// DE-BOUNCE TIMER FOR GL8 CASE STOP2 IS RAISED SWITCH OFF
GVL_CONVEYORS.GL8.CaseStop2IsRaisedTimerOff (IN := GVL_CONVEYORS.GL8.Case_Stop_Load_2_Extended_Right AND GVL_CONVEYORS.GL8.Case_Stop_Load_2_Extended_Left , PT := T#500MS);
GVL_CONVEYORS.GL8.CaseStop2IsRaisedTimerOffDoneBit := GVL_CONVEYORS.GL8.CaseStop2IsRaisedTimerOff.Q;
GVL_CONVEYORS.GL8.CaseStop2IsRaisedTimerOffElapsedTime := GVL_CONVEYORS.GL8.CaseStop2IsRaisedTimerOff.ET;
GVL_CONVEYORS.GL8.CaseStop2RaisedSwitchIsOff := GVL_CONVEYORS.GL8.CaseStop2IsRaisedTimerOffDoneBit;

END_PROGRAM

// ---- Machine System/PRGs/Conveyors/MOTOR_FAULTS.TcPOU
PROGRAM MOTOR_FAULTS
VAR
	TON_GL1_MTR: TON; // MOTOR FAULT DELAY TIMER
	TON_GL2_MTR: TON; // MOTOR FAULT DELAY TIMER
	TON_GL3_MTR: TON; // MOTOR FAULT DELAY TIMER
	TON_GL4_MTR: TON; // MOTOR FAULT DELAY TIMER
	TON_GL5A_MTR: TON; // MOTOR FAULT DELAY TIMER
	TON_GL5B_MTR: TON; // MOTOR FAULT DELAY TIMER
	TON_GL6_MTR: TON; // MOTOR FAULT DELAY TIMER
	TON_GL7_MTR: TON; // MOTOR FAULT DELAY TIMER
	TON_GL8_MTR: TON; // MOTOR FAULT DELAY TIMER
	TON_GL9_MTR: TON; // MOTOR FAULT DELAY TIMER
	TON_GL10_MTR: TON; // MOTOR FAULT DELAY TIMER
	TON_GL11_MTR: TON; // MOTOR FAULT DELAY TIMER
	
	GL1_MTR: sClearPath;
	GL2_MTR: sClearPath;
	GL3_MTR: sClearPath;
	GL4_MTR: sClearPath;
	GL5_MTR: sClearPath;
	GL6_MTR: sClearPath;
	GL7_MTR: sClearPath;
	GL8_MTR: sClearPath;
	GL9_MTR: sClearPath;
	GL10_MTR: sClearPath;
	GL11_MTR: sClearPath;
		
	
	GL1: sTransfer;
	GL2: sTransfer;
	GL3: sConveyor;
	GL4: sConveyor;
	GL5A: sConveyor;
	GL5B: sConveyor;
	GL6: sConveyor;
	GL7:sConveyor;
	GL8: sConveyor;
	GL9: sConveyor;
	GL10: sConveyor;
	GL11: sConveyor;
	GL1_RD: SRoll_Door;
	

	RUN_FWD_TO_GL6_BIT : BOOL; // GL2 OCCUPIED, GL6 REQUESTING PART, RUN TO GL6 POSITION
	RUN_FWD_TO_GL8_BIT : BOOL; // GL2 OCCUPIED, GL8 REQUESTING PART, RUN TO GL8 POSITION
	RUN_REV_TO_GL5B_BIT : BOOL; //GL2 EMPTY, GL2 REQUESTING PART, RUN TO GL5 POSITION
	MTR_FAULT_PRESET_TIME: TIME; // FAULT TIMER PRESET TO MOTOR FAULT. DEFAULT IS 1000mS.
	COUNTER_PRESET: WORD; // MAX COUNT VALUE
	
	
END_VAR
VAR // added by the converter: edge detectors and wires of the graphical bodies
    _w1 : BOOL;
END_VAR

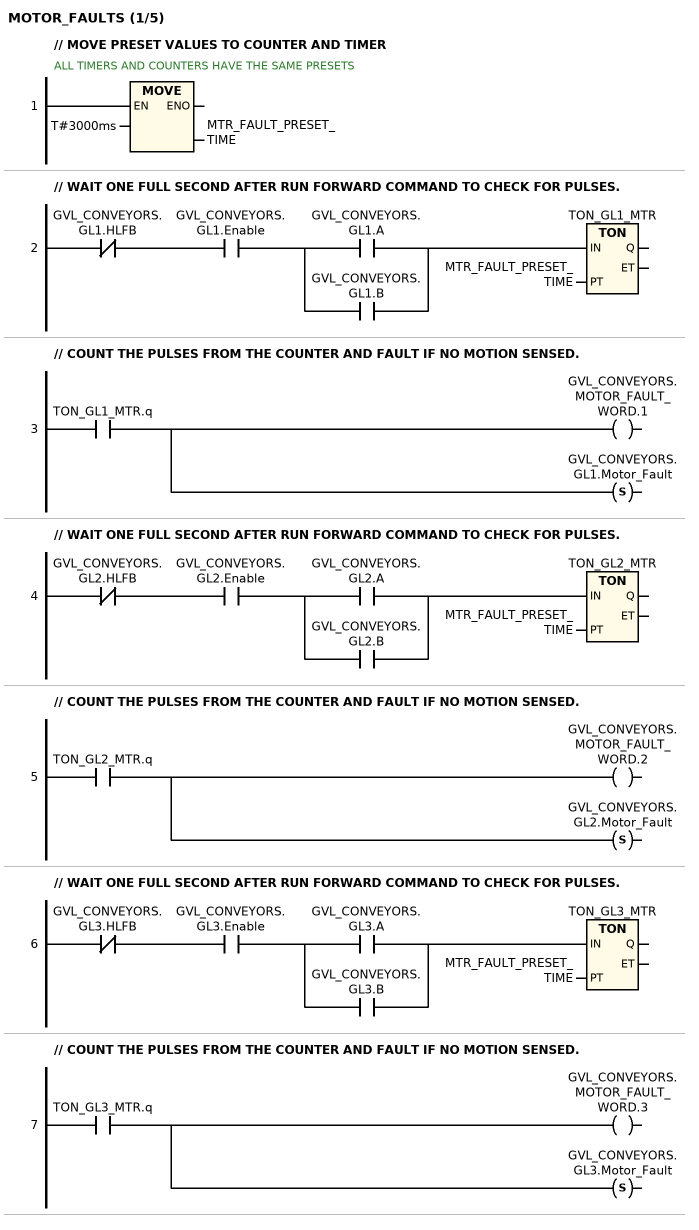
// NETWORK 1: // MOVE PRESET VALUES TO COUNTER AND TIMER
// ALL TIMERS AND COUNTERS HAVE THE SAME PRESETS
MTR_FAULT_PRESET_TIME := T#3000ms;

// NETWORK 2: // WAIT ONE FULL SECOND AFTER RUN FORWARD COMMAND TO CHECK FOR PULSES.
TON_GL1_MTR(IN := NOT GVL_CONVEYORS.GL1.HLFB AND GVL_CONVEYORS.GL1.Enable AND (GVL_CONVEYORS.GL1.A OR GVL_CONVEYORS.GL1.B), PT := MTR_FAULT_PRESET_TIME); // TON

// NETWORK 3: // COUNT THE PULSES FROM THE COUNTER AND FAULT IF NO MOTION SENSED.
GVL_CONVEYORS.MOTOR_FAULT_WORD.1 := TON_GL1_MTR.q;
GVL_CONVEYORS.GL1.Motor_Fault S= TON_GL1_MTR.q;

// NETWORK 4: // WAIT ONE FULL SECOND AFTER RUN FORWARD COMMAND TO CHECK FOR PULSES.
TON_GL2_MTR(IN := NOT GVL_CONVEYORS.GL2.HLFB AND GVL_CONVEYORS.GL2.Enable AND (GVL_CONVEYORS.GL2.A OR GVL_CONVEYORS.GL2.B), PT := MTR_FAULT_PRESET_TIME); // TON

// NETWORK 5: // COUNT THE PULSES FROM THE COUNTER AND FAULT IF NO MOTION SENSED.
GVL_CONVEYORS.MOTOR_FAULT_WORD.2 := TON_GL2_MTR.q;
GVL_CONVEYORS.GL2.Motor_Fault S= TON_GL2_MTR.q;

// NETWORK 6: // WAIT ONE FULL SECOND AFTER RUN FORWARD COMMAND TO CHECK FOR PULSES.
TON_GL3_MTR(IN := NOT GVL_CONVEYORS.GL3.HLFB AND GVL_CONVEYORS.GL3.Enable AND (GVL_CONVEYORS.GL3.A OR GVL_CONVEYORS.GL3.B), PT := MTR_FAULT_PRESET_TIME); // TON

// NETWORK 7: // COUNT THE PULSES FROM THE COUNTER AND FAULT IF NO MOTION SENSED.
GVL_CONVEYORS.MOTOR_FAULT_WORD.3 := TON_GL3_MTR.q;
GVL_CONVEYORS.GL3.Motor_Fault S= TON_GL3_MTR.q;

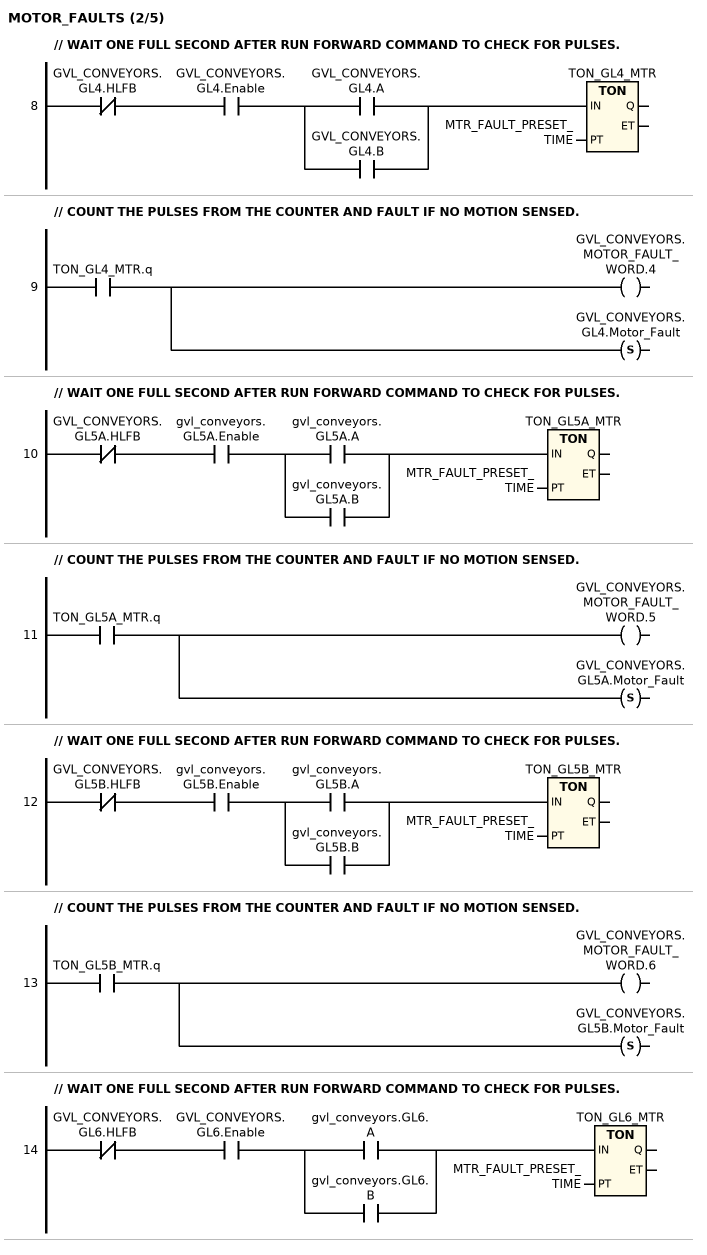
// NETWORK 8: // WAIT ONE FULL SECOND AFTER RUN FORWARD COMMAND TO CHECK FOR PULSES.
TON_GL4_MTR(IN := NOT GVL_CONVEYORS.GL4.HLFB AND GVL_CONVEYORS.GL4.Enable AND (GVL_CONVEYORS.GL4.A OR GVL_CONVEYORS.GL4.B), PT := MTR_FAULT_PRESET_TIME); // TON

// NETWORK 9: // COUNT THE PULSES FROM THE COUNTER AND FAULT IF NO MOTION SENSED.
GVL_CONVEYORS.MOTOR_FAULT_WORD.4 := TON_GL4_MTR.q;
GVL_CONVEYORS.GL4.Motor_Fault S= TON_GL4_MTR.q;

// NETWORK 10: // WAIT ONE FULL SECOND AFTER RUN FORWARD COMMAND TO CHECK FOR PULSES.
TON_GL5A_MTR(IN := NOT GVL_CONVEYORS.GL5A.HLFB AND gvl_conveyors.GL5A.Enable AND (gvl_conveyors.GL5A.A OR gvl_conveyors.GL5A.B), PT := MTR_FAULT_PRESET_TIME); // TON

// NETWORK 11: // COUNT THE PULSES FROM THE COUNTER AND FAULT IF NO MOTION SENSED.
GVL_CONVEYORS.MOTOR_FAULT_WORD.5 := TON_GL5A_MTR.q;
GVL_CONVEYORS.GL5A.Motor_Fault S= TON_GL5A_MTR.q;

// NETWORK 12: // WAIT ONE FULL SECOND AFTER RUN FORWARD COMMAND TO CHECK FOR PULSES.
TON_GL5B_MTR(IN := NOT GVL_CONVEYORS.GL5B.HLFB AND gvl_conveyors.GL5B.Enable AND (gvl_conveyors.GL5B.A OR gvl_conveyors.GL5B.B), PT := MTR_FAULT_PRESET_TIME); // TON

// NETWORK 13: // COUNT THE PULSES FROM THE COUNTER AND FAULT IF NO MOTION SENSED.
GVL_CONVEYORS.MOTOR_FAULT_WORD.6 := TON_GL5B_MTR.q;
GVL_CONVEYORS.GL5B.Motor_Fault S= TON_GL5B_MTR.q;

// NETWORK 14: // WAIT ONE FULL SECOND AFTER RUN FORWARD COMMAND TO CHECK FOR PULSES.
TON_GL6_MTR(IN := NOT GVL_CONVEYORS.GL6.HLFB AND GVL_CONVEYORS.GL6.Enable AND (gvl_conveyors.GL6.A OR gvl_conveyors.GL6.B), PT := MTR_FAULT_PRESET_TIME); // TON

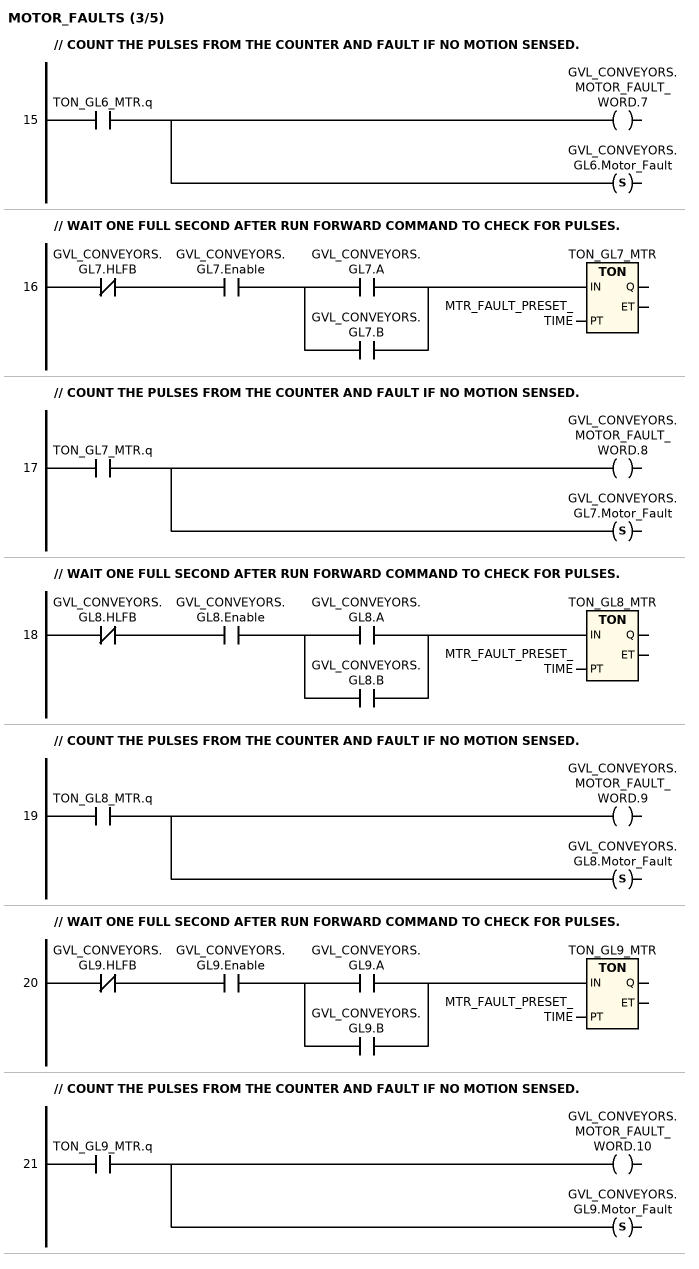
// NETWORK 15: // COUNT THE PULSES FROM THE COUNTER AND FAULT IF NO MOTION SENSED.
GVL_CONVEYORS.MOTOR_FAULT_WORD.7 := TON_GL6_MTR.q;
GVL_CONVEYORS.GL6.Motor_Fault S= TON_GL6_MTR.q;

// NETWORK 16: // WAIT ONE FULL SECOND AFTER RUN FORWARD COMMAND TO CHECK FOR PULSES.
TON_GL7_MTR(IN := NOT GVL_CONVEYORS.GL7.HLFB AND GVL_CONVEYORS.GL7.Enable AND (GVL_CONVEYORS.GL7.A OR GVL_CONVEYORS.GL7.B), PT := MTR_FAULT_PRESET_TIME); // TON

// NETWORK 17: // COUNT THE PULSES FROM THE COUNTER AND FAULT IF NO MOTION SENSED.
GVL_CONVEYORS.MOTOR_FAULT_WORD.8 := TON_GL7_MTR.q;
GVL_CONVEYORS.GL7.Motor_Fault S= TON_GL7_MTR.q;

// NETWORK 18: // WAIT ONE FULL SECOND AFTER RUN FORWARD COMMAND TO CHECK FOR PULSES.
TON_GL8_MTR(IN := NOT GVL_CONVEYORS.GL8.HLFB AND GVL_CONVEYORS.GL8.Enable AND (GVL_CONVEYORS.GL8.A OR GVL_CONVEYORS.GL8.B), PT := MTR_FAULT_PRESET_TIME); // TON

// NETWORK 19: // COUNT THE PULSES FROM THE COUNTER AND FAULT IF NO MOTION SENSED.
GVL_CONVEYORS.MOTOR_FAULT_WORD.9 := TON_GL8_MTR.q;
GVL_CONVEYORS.GL8.Motor_Fault S= TON_GL8_MTR.q;

// NETWORK 20: // WAIT ONE FULL SECOND AFTER RUN FORWARD COMMAND TO CHECK FOR PULSES.
TON_GL9_MTR(IN := NOT GVL_CONVEYORS.GL9.HLFB AND GVL_CONVEYORS.GL9.Enable AND (GVL_CONVEYORS.GL9.A OR GVL_CONVEYORS.GL9.B), PT := MTR_FAULT_PRESET_TIME); // TON

// NETWORK 21: // COUNT THE PULSES FROM THE COUNTER AND FAULT IF NO MOTION SENSED.
GVL_CONVEYORS.MOTOR_FAULT_WORD.10 := TON_GL9_MTR.q;
GVL_CONVEYORS.GL9.Motor_Fault S= TON_GL9_MTR.q;

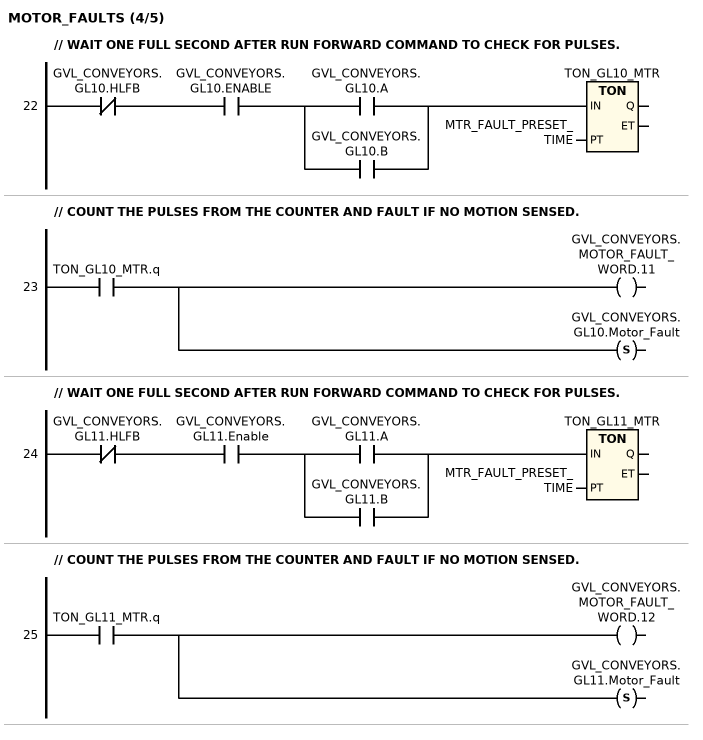
// NETWORK 22: // WAIT ONE FULL SECOND AFTER RUN FORWARD COMMAND TO CHECK FOR PULSES.
TON_GL10_MTR(IN := NOT GVL_CONVEYORS.GL10.HLFB AND GVL_CONVEYORS.GL10.ENABLE AND (GVL_CONVEYORS.GL10.A OR GVL_CONVEYORS.GL10.B), PT := MTR_FAULT_PRESET_TIME); // TON

// NETWORK 23: // COUNT THE PULSES FROM THE COUNTER AND FAULT IF NO MOTION SENSED.
GVL_CONVEYORS.MOTOR_FAULT_WORD.11 := TON_GL10_MTR.q;
GVL_CONVEYORS.GL10.Motor_Fault S= TON_GL10_MTR.q;

// NETWORK 24: // WAIT ONE FULL SECOND AFTER RUN FORWARD COMMAND TO CHECK FOR PULSES.
TON_GL11_MTR(IN := NOT GVL_CONVEYORS.GL11.HLFB AND GVL_CONVEYORS.GL11.Enable AND (GVL_CONVEYORS.GL11.A OR GVL_CONVEYORS.GL11.B), PT := MTR_FAULT_PRESET_TIME); // TON

// NETWORK 25: // COUNT THE PULSES FROM THE COUNTER AND FAULT IF NO MOTION SENSED.
GVL_CONVEYORS.MOTOR_FAULT_WORD.12 := TON_GL11_MTR.q;
GVL_CONVEYORS.GL11.Motor_Fault S= TON_GL11_MTR.q;

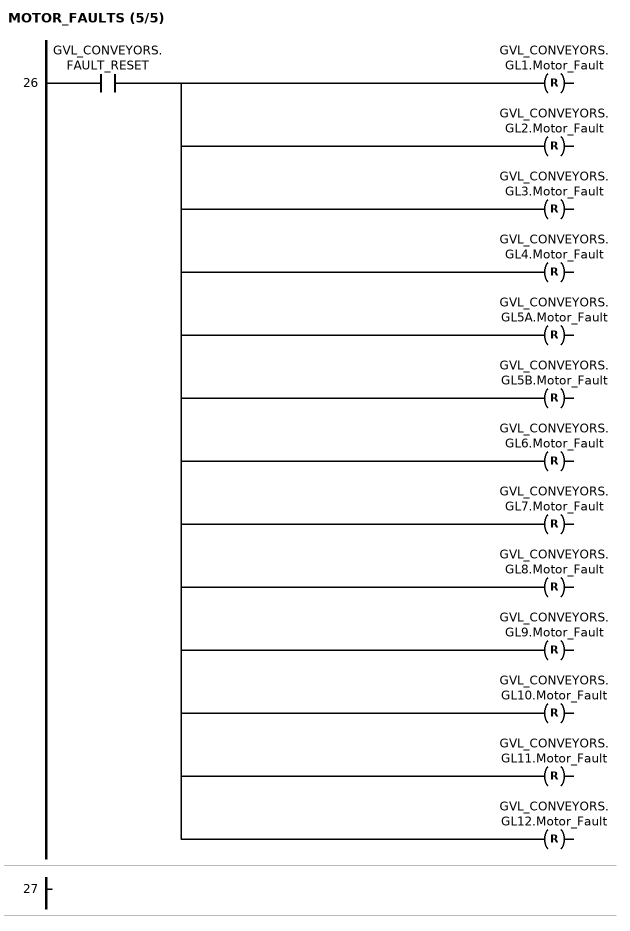
// NETWORK 26
_w1 := GVL_CONVEYORS.FAULT_RESET;
GVL_CONVEYORS.GL1.Motor_Fault R= _w1;
GVL_CONVEYORS.GL2.Motor_Fault R= _w1;
GVL_CONVEYORS.GL3.Motor_Fault R= _w1;
GVL_CONVEYORS.GL4.Motor_Fault R= _w1;
GVL_CONVEYORS.GL5A.Motor_Fault R= _w1;
GVL_CONVEYORS.GL5B.Motor_Fault R= _w1;
GVL_CONVEYORS.GL6.Motor_Fault R= _w1;
GVL_CONVEYORS.GL7.Motor_Fault R= _w1;
GVL_CONVEYORS.GL8.Motor_Fault R= _w1;
GVL_CONVEYORS.GL9.Motor_Fault R= _w1;
GVL_CONVEYORS.GL10.Motor_Fault R= _w1;
GVL_CONVEYORS.GL11.Motor_Fault R= _w1;
GVL_CONVEYORS.GL12.Motor_Fault R= _w1;

// NETWORK 27

END_PROGRAM

// ---- Machine System/PRGs/Conveyors/JAM_FAULTS.TcPOU
PROGRAM JAM_FAULTS
VAR
	TON_GL1_JAM: TON; // MOTOR FAULT DELAY TIMER
	TON_GL2_JAM: TON; // MOTOR FAULT DELAY TIMER
	TON_GL3_JAM: TON; // MOTOR FAULT DELAY TIMER
	TON_GL4_JAM: TON; // MOTOR FAULT DELAY TIMER
	TON_GL5A_JAM: TON; // MOTOR FAULT DELAY TIMER
	TON_GL5B_JAM: TON; // MOTOR FAULT DELAY TIMER
	TON_GL6_JAM: TON; // MOTOR FAULT DELAY TIMER
	TON_GL7_JAM: TON; // MOTOR FAULT DELAY TIMER
	TON_GL8_JAM: TON; // MOTOR FAULT DELAY TIMER
	TON_GL9_JAM: TON; // MOTOR FAULT DELAY TIMER
	TON_GL10_JAM: TON; // MOTOR FAULT DELAY TIMER
	TON_GL11_JAM: TON; // MOTOR FAULT DELAY TIMER
	FAULT_PRESET_TIME: time;
	
			
	GL1: sTransfer;
	GL2: sTransfer;
	GL3: sConveyor;
	GL4: sConveyor;
	GL5: sConveyor;
	GL6: sConveyor;
	GL7:sConveyor;
	GL8: sConveyor;
	GL9: sConveyor;
	GL10: sConveyor;
	GL11: sTransfer;
	GL1_RD: SRoll_Door;
		
END_VAR
VAR // added by the converter: edge detectors and wires of the graphical bodies
    _w1 : BOOL;
END_VAR

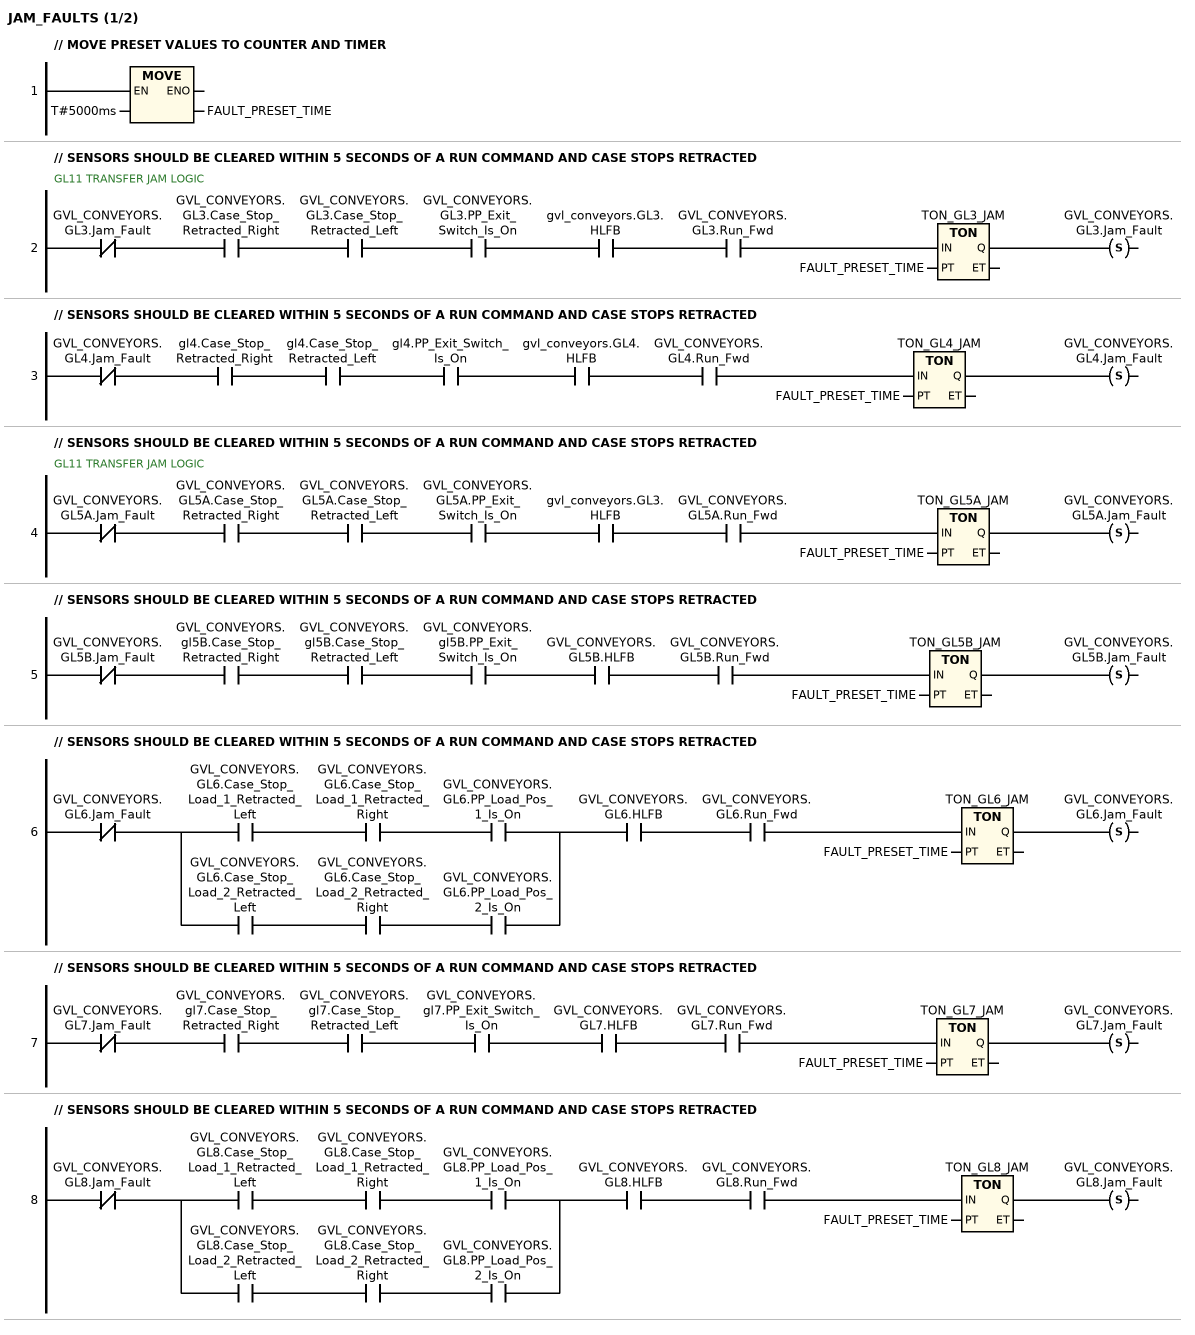
// NETWORK 1: // MOVE PRESET VALUES TO COUNTER AND TIMER
FAULT_PRESET_TIME := T#5000ms;

// NETWORK 2: // SENSORS SHOULD BE CLEARED WITHIN 5 SECONDS OF A RUN COMMAND AND CASE STOPS RETRACTED
// GL11 TRANSFER JAM LOGIC
TON_GL3_JAM(IN := NOT GVL_CONVEYORS.GL3.Jam_Fault AND GVL_CONVEYORS.GL3.Case_Stop_Retracted_Right AND GVL_CONVEYORS.GL3.Case_Stop_Retracted_Left AND GVL_CONVEYORS.GL3.PP_Exit_Switch_Is_On AND gvl_conveyors.GL3.HLFB AND GVL_CONVEYORS.GL3.Run_Fwd, PT := FAULT_PRESET_TIME); // TON
GVL_CONVEYORS.GL3.Jam_Fault S= TON_GL3_JAM.Q;

// NETWORK 3: // SENSORS SHOULD BE CLEARED WITHIN 5 SECONDS OF A RUN COMMAND AND CASE STOPS RETRACTED
TON_GL4_JAM(IN := NOT GVL_CONVEYORS.GL4.Jam_Fault AND gl4.Case_Stop_Retracted_Right AND gl4.Case_Stop_Retracted_Left AND gl4.PP_Exit_Switch_Is_On AND gvl_conveyors.GL4.HLFB AND GVL_CONVEYORS.GL4.Run_Fwd, PT := FAULT_PRESET_TIME); // TON
GVL_CONVEYORS.GL4.Jam_Fault S= TON_GL4_JAM.Q;

// NETWORK 4: // SENSORS SHOULD BE CLEARED WITHIN 5 SECONDS OF A RUN COMMAND AND CASE STOPS RETRACTED
// GL11 TRANSFER JAM LOGIC
TON_GL5A_JAM(IN := NOT GVL_CONVEYORS.GL5A.Jam_Fault AND GVL_CONVEYORS.GL5A.Case_Stop_Retracted_Right AND GVL_CONVEYORS.GL5A.Case_Stop_Retracted_Left AND GVL_CONVEYORS.GL5A.PP_Exit_Switch_Is_On AND gvl_conveyors.GL3.HLFB AND GVL_CONVEYORS.GL5A.Run_Fwd, PT := FAULT_PRESET_TIME); // TON
GVL_CONVEYORS.GL5A.Jam_Fault S= TON_GL5A_JAM.Q;

// NETWORK 5: // SENSORS SHOULD BE CLEARED WITHIN 5 SECONDS OF A RUN COMMAND AND CASE STOPS RETRACTED
TON_GL5B_JAM(IN := NOT GVL_CONVEYORS.GL5B.Jam_Fault AND GVL_CONVEYORS.gl5B.Case_Stop_Retracted_Right AND GVL_CONVEYORS.gl5B.Case_Stop_Retracted_Left AND GVL_CONVEYORS.gl5B.PP_Exit_Switch_Is_On AND GVL_CONVEYORS.GL5B.HLFB AND GVL_CONVEYORS.GL5B.Run_Fwd, PT := FAULT_PRESET_TIME); // TON
GVL_CONVEYORS.GL5B.Jam_Fault S= TON_GL5B_JAM.Q;

// NETWORK 6: // SENSORS SHOULD BE CLEARED WITHIN 5 SECONDS OF A RUN COMMAND AND CASE STOPS RETRACTED
TON_GL6_JAM(IN := NOT GVL_CONVEYORS.GL6.Jam_Fault AND (GVL_CONVEYORS.GL6.Case_Stop_Load_1_Retracted_Left AND GVL_CONVEYORS.GL6.Case_Stop_Load_1_Retracted_Right AND GVL_CONVEYORS.GL6.PP_Load_Pos_1_Is_On OR GVL_CONVEYORS.GL6.Case_Stop_Load_2_Retracted_Left AND GVL_CONVEYORS.GL6.Case_Stop_Load_2_Retracted_Right AND GVL_CONVEYORS.GL6.PP_Load_Pos_2_Is_On) AND GVL_CONVEYORS.GL6.HLFB AND GVL_CONVEYORS.GL6.Run_Fwd, PT := FAULT_PRESET_TIME); // TON
GVL_CONVEYORS.GL6.Jam_Fault S= TON_GL6_JAM.Q;

// NETWORK 7: // SENSORS SHOULD BE CLEARED WITHIN 5 SECONDS OF A RUN COMMAND AND CASE STOPS RETRACTED
TON_GL7_JAM(IN := NOT GVL_CONVEYORS.GL7.Jam_Fault AND GVL_CONVEYORS.gl7.Case_Stop_Retracted_Right AND GVL_CONVEYORS.gl7.Case_Stop_Retracted_Left AND GVL_CONVEYORS.gl7.PP_Exit_Switch_Is_On AND GVL_CONVEYORS.GL7.HLFB AND GVL_CONVEYORS.GL7.Run_Fwd, PT := FAULT_PRESET_TIME); // TON
GVL_CONVEYORS.GL7.Jam_Fault S= TON_GL7_JAM.Q;

// NETWORK 8: // SENSORS SHOULD BE CLEARED WITHIN 5 SECONDS OF A RUN COMMAND AND CASE STOPS RETRACTED
TON_GL8_JAM(IN := NOT GVL_CONVEYORS.GL8.Jam_Fault AND (GVL_CONVEYORS.GL8.Case_Stop_Load_1_Retracted_Left AND GVL_CONVEYORS.GL8.Case_Stop_Load_1_Retracted_Right AND GVL_CONVEYORS.GL8.PP_Load_Pos_1_Is_On OR GVL_CONVEYORS.GL8.Case_Stop_Load_2_Retracted_Left AND GVL_CONVEYORS.GL8.Case_Stop_Load_2_Retracted_Right AND GVL_CONVEYORS.GL8.PP_Load_Pos_2_Is_On) AND GVL_CONVEYORS.GL8.HLFB AND GVL_CONVEYORS.GL8.Run_Fwd, PT := FAULT_PRESET_TIME); // TON
GVL_CONVEYORS.GL8.Jam_Fault S= TON_GL8_JAM.Q;

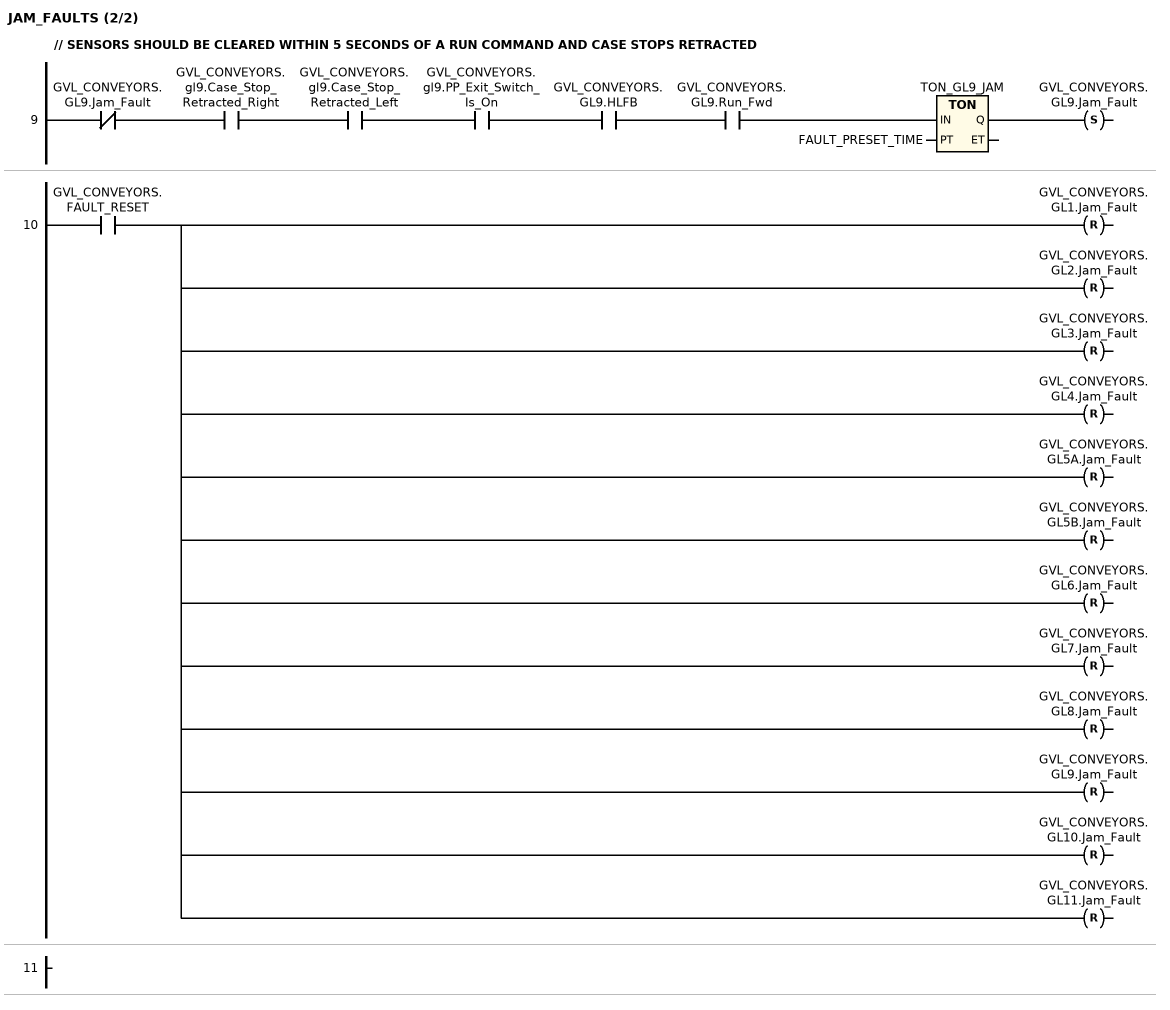
// NETWORK 9: // SENSORS SHOULD BE CLEARED WITHIN 5 SECONDS OF A RUN COMMAND AND CASE STOPS RETRACTED
TON_GL9_JAM(IN := NOT GVL_CONVEYORS.GL9.Jam_Fault AND GVL_CONVEYORS.gl9.Case_Stop_Retracted_Right AND GVL_CONVEYORS.gl9.Case_Stop_Retracted_Left AND GVL_CONVEYORS.gl9.PP_Exit_Switch_Is_On AND GVL_CONVEYORS.GL9.HLFB AND GVL_CONVEYORS.GL9.Run_Fwd, PT := FAULT_PRESET_TIME); // TON
GVL_CONVEYORS.GL9.Jam_Fault S= TON_GL9_JAM.Q;

// NETWORK 10
_w1 := GVL_CONVEYORS.FAULT_RESET;
GVL_CONVEYORS.GL1.Jam_Fault R= _w1;
GVL_CONVEYORS.GL2.Jam_Fault R= _w1;
GVL_CONVEYORS.GL3.Jam_Fault R= _w1;
GVL_CONVEYORS.GL4.Jam_Fault R= _w1;
GVL_CONVEYORS.GL5A.Jam_Fault R= _w1;
GVL_CONVEYORS.GL5B.Jam_Fault R= _w1;
GVL_CONVEYORS.GL6.Jam_Fault R= _w1;
GVL_CONVEYORS.GL7.Jam_Fault R= _w1;
GVL_CONVEYORS.GL8.Jam_Fault R= _w1;
GVL_CONVEYORS.GL9.Jam_Fault R= _w1;
GVL_CONVEYORS.GL10.Jam_Fault R= _w1;
GVL_CONVEYORS.GL11.Jam_Fault R= _w1;

// NETWORK 11

END_PROGRAM

// ---- Machine System/PRGs/Conveyors/OUTPUTS.TcPOU
PROGRAM OUTPUTS
VAR
	C6_K1_SAFETY_CONTACTOR AT %Q*: BOOL; // 
	C6_K2_SAFETY_CONTACTOR AT %Q*: BOOL; // 
	C7_K1_SAFETY_CONTACTOR AT %Q*: BOOL; // 
	C7_K2_SAFETY_CONTACTOR AT %Q*: BOOL; // 	



KIRK_BIT: BOOL;
BTEST :BOOL;
	
//GL4: sConveyor;
	

//GL5A:sConveyor;
	
	
//GL5B: sConveyor;
//GL6: sConveyor;
//GL7: sConveyor;
//GL8: sConveyor;
//GL9: sConveyor;
	
END_VAR

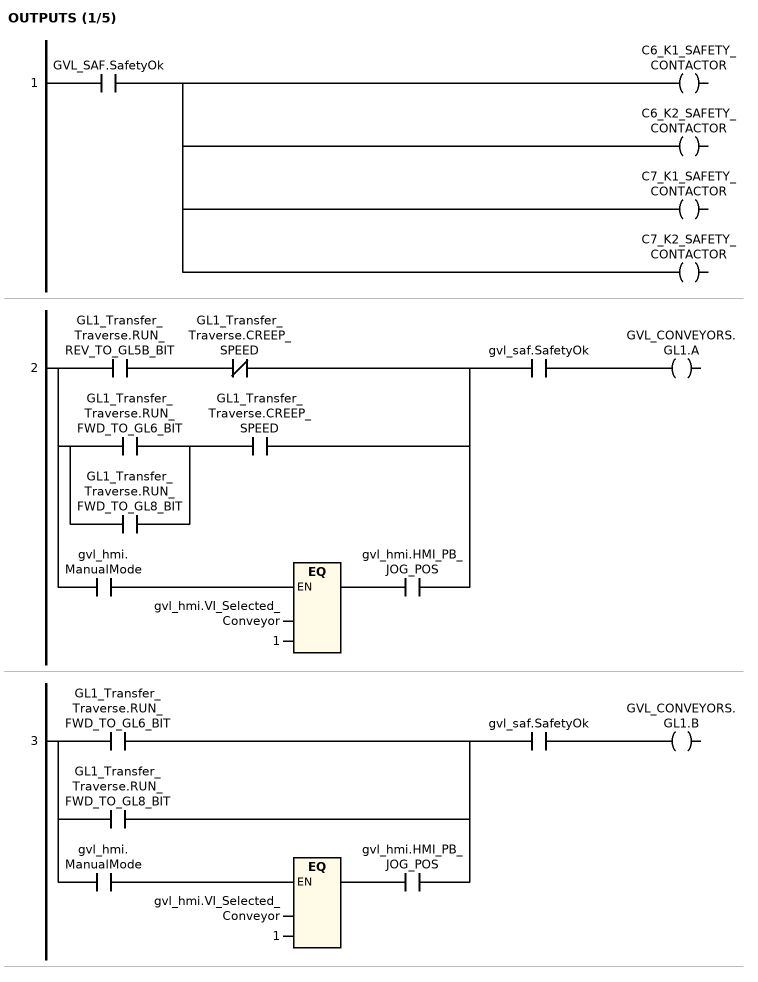
// NETWORK 1
C6_K1_SAFETY_CONTACTOR := GVL_SAF.SafetyOk;
C6_K2_SAFETY_CONTACTOR := GVL_SAF.SafetyOk;
C7_K1_SAFETY_CONTACTOR := GVL_SAF.SafetyOk;
C7_K2_SAFETY_CONTACTOR := GVL_SAF.SafetyOk;

// NETWORK 2
GVL_CONVEYORS.GL1.A := (GL1_Transfer_Traverse.RUN_REV_TO_GL5B_BIT AND NOT GL1_Transfer_Traverse.CREEP_SPEED OR (GL1_Transfer_Traverse.RUN_FWD_TO_GL6_BIT OR GL1_Transfer_Traverse.RUN_FWD_TO_GL8_BIT) AND GL1_Transfer_Traverse.CREEP_SPEED OR (gvl_hmi.ManualMode AND gvl_hmi.VI_Selected_Conveyor = 1) AND gvl_hmi.HMI_PB_JOG_POS) AND gvl_saf.SafetyOk;

// NETWORK 3
GVL_CONVEYORS.GL1.B := (GL1_Transfer_Traverse.RUN_FWD_TO_GL6_BIT OR GL1_Transfer_Traverse.RUN_FWD_TO_GL8_BIT OR (gvl_hmi.ManualMode AND gvl_hmi.VI_Selected_Conveyor = 1) AND gvl_hmi.HMI_PB_JOG_POS) AND gvl_saf.SafetyOk;

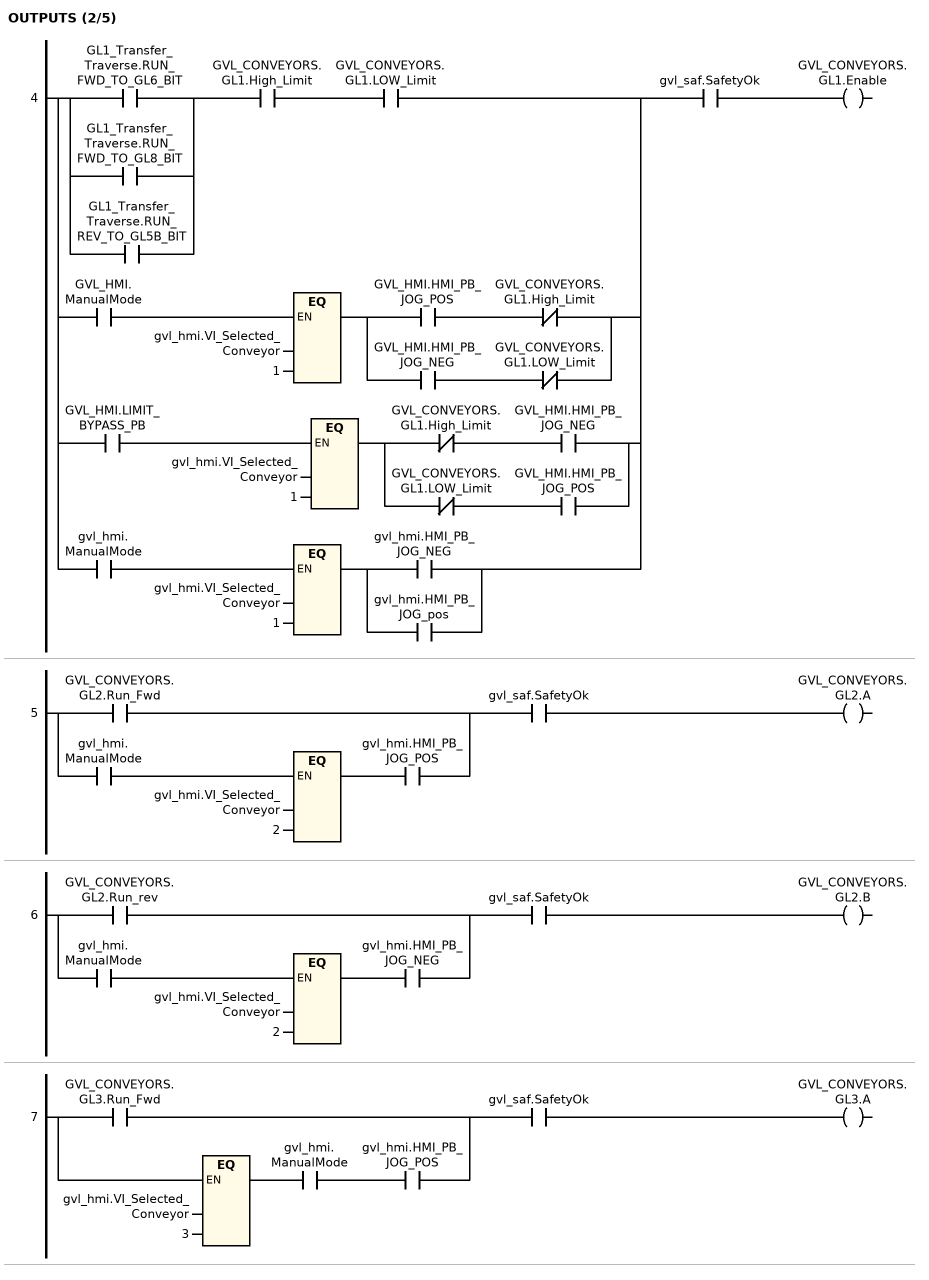
// NETWORK 4
GVL_CONVEYORS.GL1.Enable := ((GL1_Transfer_Traverse.RUN_FWD_TO_GL6_BIT OR GL1_Transfer_Traverse.RUN_FWD_TO_GL8_BIT OR GL1_Transfer_Traverse.RUN_REV_TO_GL5B_BIT) AND GVL_CONVEYORS.GL1.High_Limit AND GVL_CONVEYORS.GL1.LOW_Limit OR (GVL_HMI.ManualMode AND gvl_hmi.VI_Selected_Conveyor = 1) AND (GVL_HMI.HMI_PB_JOG_POS AND NOT GVL_CONVEYORS.GL1.High_Limit OR GVL_HMI.HMI_PB_JOG_NEG AND NOT GVL_CONVEYORS.GL1.LOW_Limit) OR (GVL_HMI.LIMIT_BYPASS_PB AND gvl_hmi.VI_Selected_Conveyor = 1) AND (NOT GVL_CONVEYORS.GL1.High_Limit AND GVL_HMI.HMI_PB_JOG_NEG OR NOT GVL_CONVEYORS.GL1.LOW_Limit AND GVL_HMI.HMI_PB_JOG_POS) OR (gvl_hmi.ManualMode AND gvl_hmi.VI_Selected_Conveyor = 1) AND (gvl_hmi.HMI_PB_JOG_NEG OR gvl_hmi.HMI_PB_JOG_pos)) AND gvl_saf.SafetyOk;

// NETWORK 5
GVL_CONVEYORS.GL2.A := (GVL_CONVEYORS.GL2.Run_Fwd OR (gvl_hmi.ManualMode AND gvl_hmi.VI_Selected_Conveyor = 2) AND gvl_hmi.HMI_PB_JOG_POS) AND gvl_saf.SafetyOk;

// NETWORK 6
GVL_CONVEYORS.GL2.B := (GVL_CONVEYORS.GL2.Run_rev OR (gvl_hmi.ManualMode AND gvl_hmi.VI_Selected_Conveyor = 2) AND gvl_hmi.HMI_PB_JOG_NEG) AND gvl_saf.SafetyOk;

// NETWORK 7
GVL_CONVEYORS.GL3.A := (GVL_CONVEYORS.GL3.Run_Fwd OR gvl_hmi.VI_Selected_Conveyor = 3 AND gvl_hmi.ManualMode AND gvl_hmi.HMI_PB_JOG_POS) AND gvl_saf.SafetyOk;

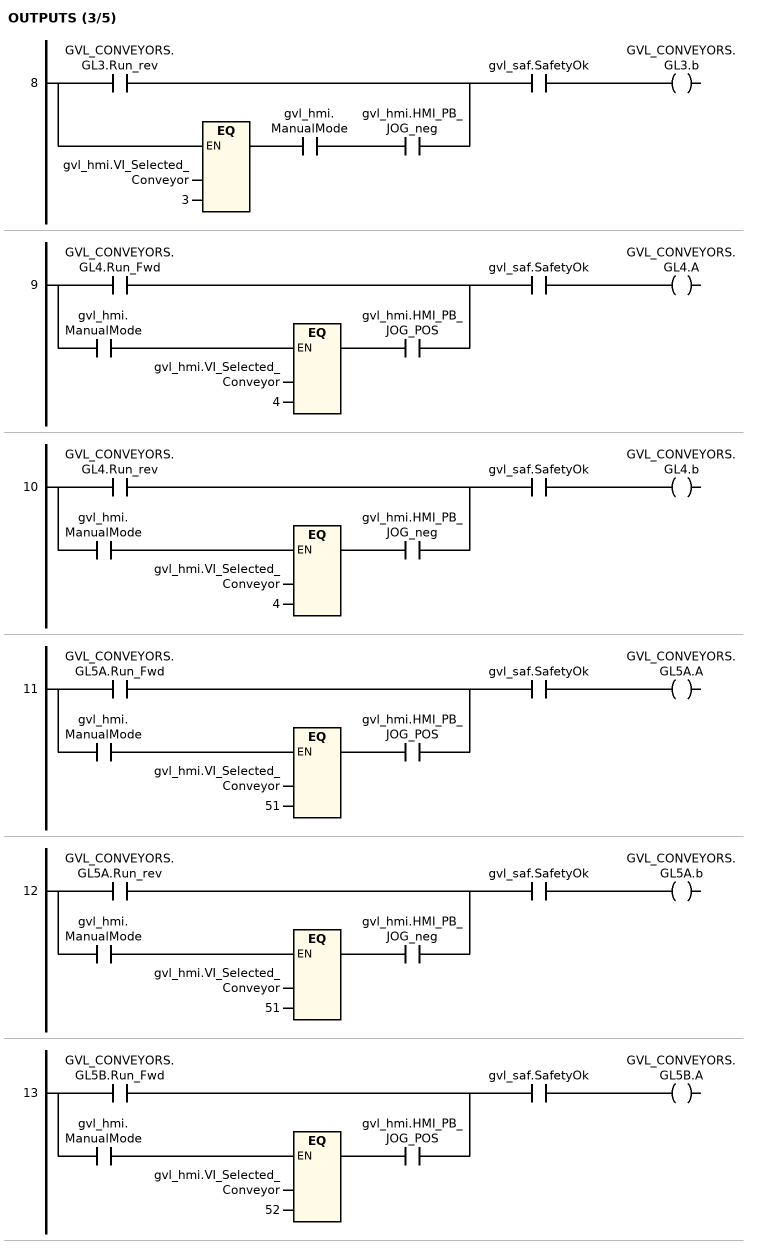
// NETWORK 8
GVL_CONVEYORS.GL3.b := (GVL_CONVEYORS.GL3.Run_rev OR gvl_hmi.VI_Selected_Conveyor = 3 AND gvl_hmi.ManualMode AND gvl_hmi.HMI_PB_JOG_neg) AND gvl_saf.SafetyOk;

// NETWORK 9
GVL_CONVEYORS.GL4.A := (GVL_CONVEYORS.GL4.Run_Fwd OR (gvl_hmi.ManualMode AND gvl_hmi.VI_Selected_Conveyor = 4) AND gvl_hmi.HMI_PB_JOG_POS) AND gvl_saf.SafetyOk;

// NETWORK 10
GVL_CONVEYORS.GL4.b := (GVL_CONVEYORS.GL4.Run_rev OR (gvl_hmi.ManualMode AND gvl_hmi.VI_Selected_Conveyor = 4) AND gvl_hmi.HMI_PB_JOG_neg) AND gvl_saf.SafetyOk;

// NETWORK 11
GVL_CONVEYORS.GL5A.A := (GVL_CONVEYORS.GL5A.Run_Fwd OR (gvl_hmi.ManualMode AND gvl_hmi.VI_Selected_Conveyor = 51) AND gvl_hmi.HMI_PB_JOG_POS) AND gvl_saf.SafetyOk;

// NETWORK 12
GVL_CONVEYORS.GL5A.b := (GVL_CONVEYORS.GL5A.Run_rev OR (gvl_hmi.ManualMode AND gvl_hmi.VI_Selected_Conveyor = 51) AND gvl_hmi.HMI_PB_JOG_neg) AND gvl_saf.SafetyOk;

// NETWORK 13
GVL_CONVEYORS.GL5B.A := (GVL_CONVEYORS.GL5B.Run_Fwd OR (gvl_hmi.ManualMode AND gvl_hmi.VI_Selected_Conveyor = 52) AND gvl_hmi.HMI_PB_JOG_POS) AND gvl_saf.SafetyOk;

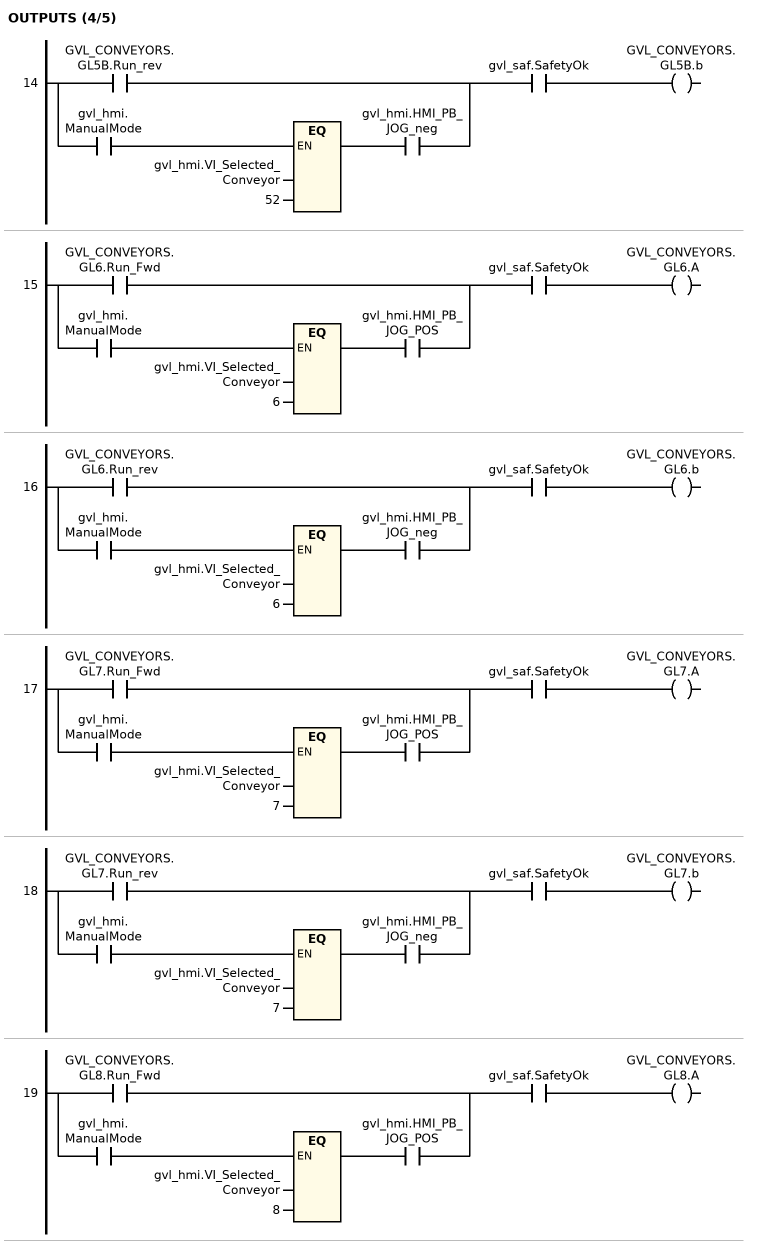
// NETWORK 14
GVL_CONVEYORS.GL5B.b := (GVL_CONVEYORS.GL5B.Run_rev OR (gvl_hmi.ManualMode AND gvl_hmi.VI_Selected_Conveyor = 52) AND gvl_hmi.HMI_PB_JOG_neg) AND gvl_saf.SafetyOk;

// NETWORK 15
GVL_CONVEYORS.GL6.A := (GVL_CONVEYORS.GL6.Run_Fwd OR (gvl_hmi.ManualMode AND gvl_hmi.VI_Selected_Conveyor = 6) AND gvl_hmi.HMI_PB_JOG_POS) AND gvl_saf.SafetyOk;

// NETWORK 16
GVL_CONVEYORS.GL6.b := (GVL_CONVEYORS.GL6.Run_rev OR (gvl_hmi.ManualMode AND gvl_hmi.VI_Selected_Conveyor = 6) AND gvl_hmi.HMI_PB_JOG_neg) AND gvl_saf.SafetyOk;

// NETWORK 17
GVL_CONVEYORS.GL7.A := (GVL_CONVEYORS.GL7.Run_Fwd OR (gvl_hmi.ManualMode AND gvl_hmi.VI_Selected_Conveyor = 7) AND gvl_hmi.HMI_PB_JOG_POS) AND gvl_saf.SafetyOk;

// NETWORK 18
GVL_CONVEYORS.GL7.b := (GVL_CONVEYORS.GL7.Run_rev OR (gvl_hmi.ManualMode AND gvl_hmi.VI_Selected_Conveyor = 7) AND gvl_hmi.HMI_PB_JOG_neg) AND gvl_saf.SafetyOk;

// NETWORK 19
GVL_CONVEYORS.GL8.A := (GVL_CONVEYORS.GL8.Run_Fwd OR (gvl_hmi.ManualMode AND gvl_hmi.VI_Selected_Conveyor = 8) AND gvl_hmi.HMI_PB_JOG_POS) AND gvl_saf.SafetyOk;

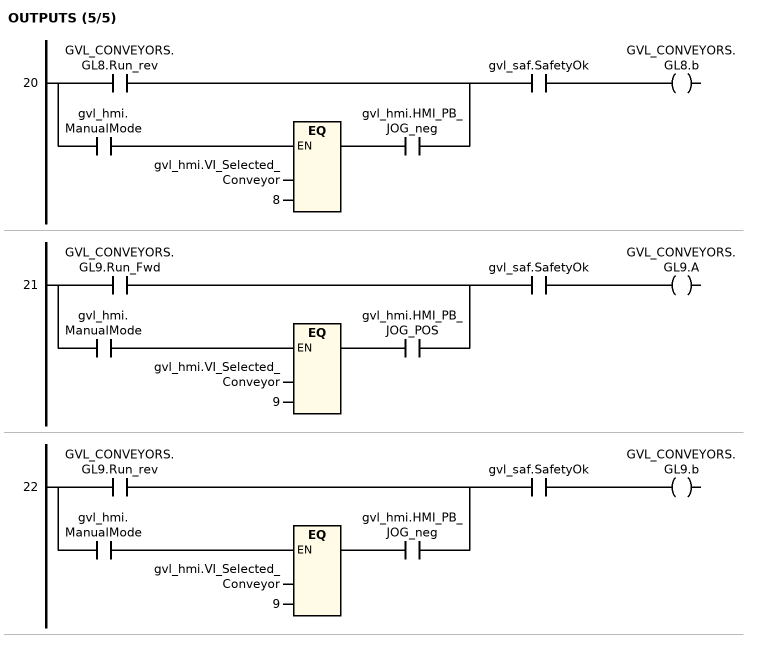
// NETWORK 20
GVL_CONVEYORS.GL8.b := (GVL_CONVEYORS.GL8.Run_rev OR (gvl_hmi.ManualMode AND gvl_hmi.VI_Selected_Conveyor = 8) AND gvl_hmi.HMI_PB_JOG_neg) AND gvl_saf.SafetyOk;

// NETWORK 21
GVL_CONVEYORS.GL9.A := (GVL_CONVEYORS.GL9.Run_Fwd OR (gvl_hmi.ManualMode AND gvl_hmi.VI_Selected_Conveyor = 9) AND gvl_hmi.HMI_PB_JOG_POS) AND gvl_saf.SafetyOk;

// NETWORK 22
GVL_CONVEYORS.GL9.b := (GVL_CONVEYORS.GL9.Run_rev OR (gvl_hmi.ManualMode AND gvl_hmi.VI_Selected_Conveyor = 9) AND gvl_hmi.HMI_PB_JOG_neg) AND gvl_saf.SafetyOk;

END_PROGRAM

// ---- Machine System/PRGs/Conveyors/GL1_Transfer_Traverse.TcPOU
PROGRAM GL1_Transfer_Traverse
VAR
	TON_GL1_MTR: TON; // MOTOR FAULT DELAY TIMER
	GL1_MTR: sClearPath;
	GL1_Pulses: INT; // CURRENT PULSE COUNT VALUE
	GL1_Pulse_Counter: CTU; // GL1 MOTOR PULSE COUNTER
	TEST: BOOL;
	GL1_RD: SRoll_Door;
	GL1_PULSE_RESET : BOOL; // RESET THE PULSE COUNTER WHEN COUNTER REACHES PRESET VALUE
	RUN_FWD_TO_GL6_BIT : BOOL; // GL2 OCCUPIED, GL6 REQUESTING PART, RUN TO GL6 POSITION
	RUN_FWD_TO_GL8_BIT : BOOL; // GL2 OCCUPIED, GL8 REQUESTING PART, RUN TO GL8 POSITION
	RUN_REV_TO_GL5B_BIT : BOOL; //GL2 EMPTY, GL2 REQUESTING PART, RUN TO GL5 POSITION
	FAULT_PRESET_TIME: TIME; // FAULT TIMER PRESET TO MOTOR FAULT. DEFAULT IS 1000mS.
	COUNTER_PRESET: WORD; // MAX COUNT VALUE
	TON_GL1_MTR_DONE: BOOL; // TIMER DONE BIT
	KIRK_BIT: BOOL;
	KIRK_BIT2: BOOL;
	KIRK_BIT3: BOOL;
	HI_SPEED: BOOL; // RUN AT HI SPPED TILL FIRST PROX SEEN
	CREEP_SPEED: BOOL; // RUN AT CREEP SPEED TILL SECOND PROX SEEN
	PROX_1_SEEN_AT_GL6: BOOL; // FIRST PROX MADE
	PROX_2_SEEN_AT_GL6: BOOL; // SECOND PROX MADE
	PROX_1_SEEN_AT_GL8: BOOL; // FIRST PROX MADE
	PROX_2_SEEN_AT_GL8: BOOL; // SECOND PROX MADE
	PROX_1_SEEN_AT_GL5B: BOOL; // FIRST PROX MADE
	PROX_2_SEEN_AT_GL5B: BOOL; // SECOND PROX MADE
	TON_CREEP_DELAY: TON; // DELAY CREEP SPEED
	GL6_ENTRY_FTRIG:  F_TRIG;
	GL8_ENTRY_FTRIG:  F_TRIG;
	SwitchFaultTimer: ton;
	SwitchFault: BOOL;
	SwitchTimeElapsed: TIME;
	
END_VAR
VAR // added by the converter: edge detectors and wires of the graphical bodies
    _rt1, _rt2 : R_TRIG;
    _w1, _w2, _w3, _w4, _w5, _w6 : BOOL;
END_VAR

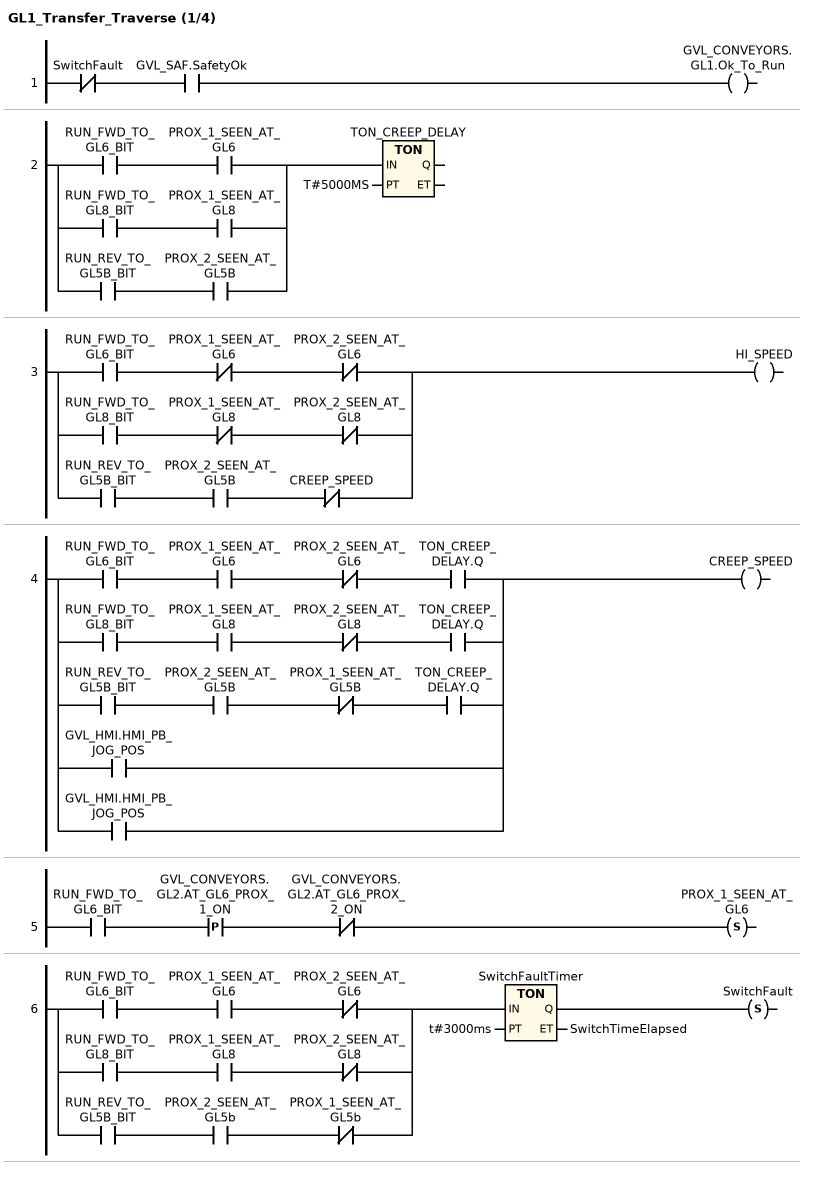
// NETWORK 1
GVL_CONVEYORS.GL1.Ok_To_Run := NOT SwitchFault AND GVL_SAF.SafetyOk;

// NETWORK 2
TON_CREEP_DELAY(IN := RUN_FWD_TO_GL6_BIT AND PROX_1_SEEN_AT_GL6 OR RUN_FWD_TO_GL8_BIT AND PROX_1_SEEN_AT_GL8 OR RUN_REV_TO_GL5B_BIT AND PROX_2_SEEN_AT_GL5B, PT := T#5000MS); // TON

// NETWORK 3
HI_SPEED := RUN_FWD_TO_GL6_BIT AND NOT PROX_1_SEEN_AT_GL6 AND NOT PROX_2_SEEN_AT_GL6 OR RUN_FWD_TO_GL8_BIT AND NOT PROX_1_SEEN_AT_GL8 AND NOT PROX_2_SEEN_AT_GL8 OR RUN_REV_TO_GL5B_BIT AND PROX_2_SEEN_AT_GL5B AND NOT CREEP_SPEED;

// NETWORK 4
CREEP_SPEED := RUN_FWD_TO_GL6_BIT AND PROX_1_SEEN_AT_GL6 AND NOT PROX_2_SEEN_AT_GL6 AND TON_CREEP_DELAY.Q OR RUN_FWD_TO_GL8_BIT AND PROX_1_SEEN_AT_GL8 AND NOT PROX_2_SEEN_AT_GL8 AND TON_CREEP_DELAY.Q OR RUN_REV_TO_GL5B_BIT AND PROX_2_SEEN_AT_GL5B AND NOT PROX_1_SEEN_AT_GL5B AND TON_CREEP_DELAY.Q OR GVL_HMI.HMI_PB_JOG_POS OR GVL_HMI.HMI_PB_JOG_POS;

// NETWORK 5
_rt1(CLK := GVL_CONVEYORS.GL2.AT_GL6_PROX_1_ON);
PROX_1_SEEN_AT_GL6 S= RUN_FWD_TO_GL6_BIT AND _rt1.Q AND NOT GVL_CONVEYORS.GL2.AT_GL6_PROX_2_ON;

// NETWORK 6
SwitchFaultTimer(
    IN := RUN_FWD_TO_GL6_BIT AND PROX_1_SEEN_AT_GL6 AND NOT PROX_2_SEEN_AT_GL6 OR RUN_FWD_TO_GL8_BIT AND PROX_1_SEEN_AT_GL8 AND NOT PROX_2_SEEN_AT_GL8 OR RUN_REV_TO_GL5B_BIT AND PROX_2_SEEN_AT_GL5b AND NOT PROX_1_SEEN_AT_GL5b,
    PT := t#3000ms,
    ET => SwitchTimeElapsed); // TON
SwitchFault S= SwitchFaultTimer.Q;

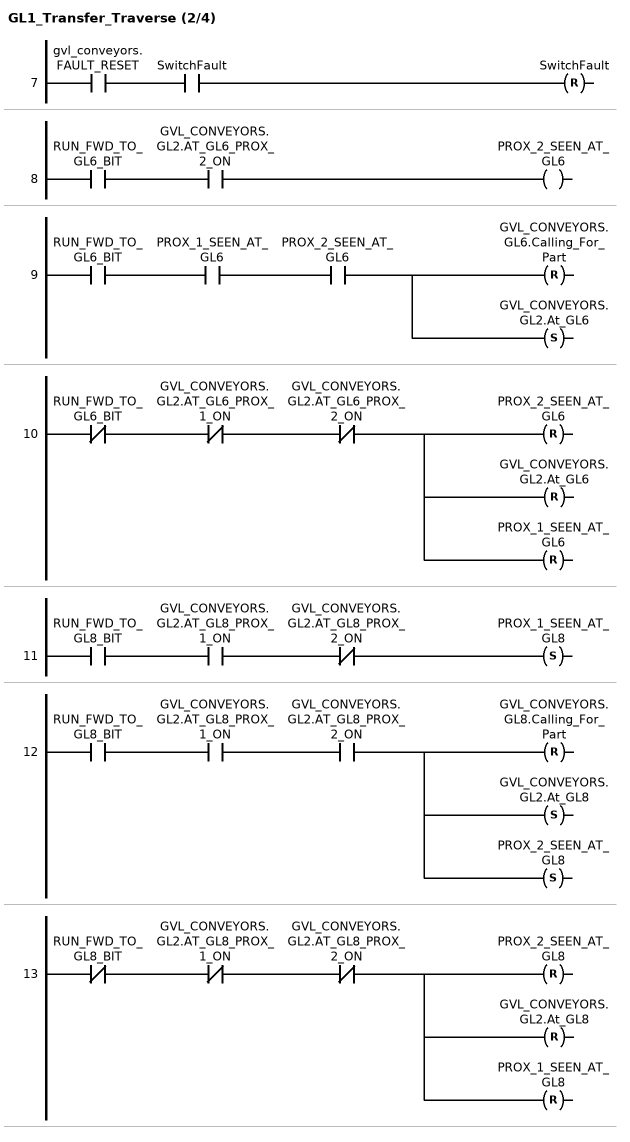
// NETWORK 7
SwitchFault R= gvl_conveyors.FAULT_RESET AND SwitchFault;

// NETWORK 8
PROX_2_SEEN_AT_GL6 := RUN_FWD_TO_GL6_BIT AND GVL_CONVEYORS.GL2.AT_GL6_PROX_2_ON;

// NETWORK 9
_w1 := RUN_FWD_TO_GL6_BIT AND PROX_1_SEEN_AT_GL6 AND PROX_2_SEEN_AT_GL6;
GVL_CONVEYORS.GL6.Calling_For_Part R= _w1;
GVL_CONVEYORS.GL2.At_GL6 S= _w1;

// NETWORK 10
_w2 := NOT RUN_FWD_TO_GL6_BIT AND NOT GVL_CONVEYORS.GL2.AT_GL6_PROX_1_ON AND NOT GVL_CONVEYORS.GL2.AT_GL6_PROX_2_ON;
PROX_2_SEEN_AT_GL6 R= _w2;
GVL_CONVEYORS.GL2.At_GL6 R= _w2;
PROX_1_SEEN_AT_GL6 R= _w2;

// NETWORK 11
PROX_1_SEEN_AT_GL8 S= RUN_FWD_TO_GL8_BIT AND GVL_CONVEYORS.GL2.AT_GL8_PROX_1_ON AND NOT GVL_CONVEYORS.GL2.AT_GL8_PROX_2_ON;

// NETWORK 12
_w3 := RUN_FWD_TO_GL8_BIT AND GVL_CONVEYORS.GL2.AT_GL8_PROX_1_ON AND GVL_CONVEYORS.GL2.AT_GL8_PROX_2_ON;
GVL_CONVEYORS.GL8.Calling_For_Part R= _w3;
GVL_CONVEYORS.GL2.At_GL8 S= _w3;
PROX_2_SEEN_AT_GL8 S= _w3;

// NETWORK 13
_w4 := NOT RUN_FWD_TO_GL8_BIT AND NOT GVL_CONVEYORS.GL2.AT_GL8_PROX_1_ON AND NOT GVL_CONVEYORS.GL2.AT_GL8_PROX_2_ON;
PROX_2_SEEN_AT_GL8 R= _w4;
GVL_CONVEYORS.GL2.At_GL8 R= _w4;
PROX_1_SEEN_AT_GL8 R= _w4;

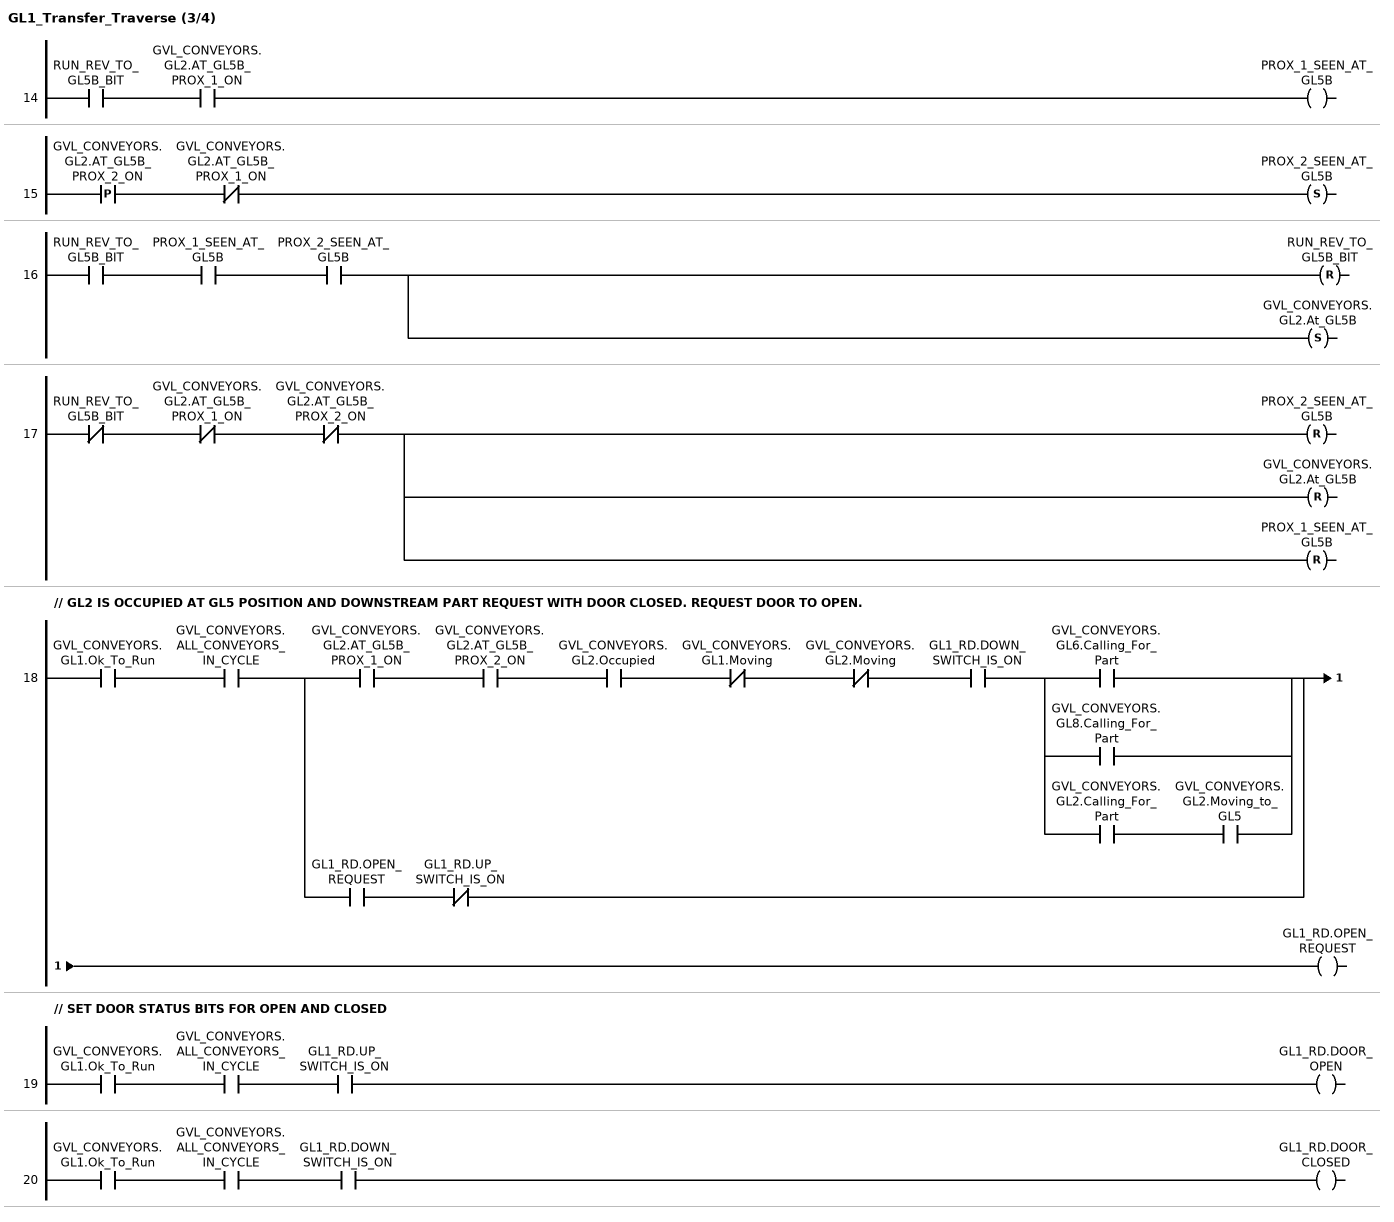
// NETWORK 14
PROX_1_SEEN_AT_GL5B := RUN_REV_TO_GL5B_BIT AND GVL_CONVEYORS.GL2.AT_GL5B_PROX_1_ON;

// NETWORK 15
_rt2(CLK := GVL_CONVEYORS.GL2.AT_GL5B_PROX_2_ON);
PROX_2_SEEN_AT_GL5B S= _rt2.Q AND NOT GVL_CONVEYORS.GL2.AT_GL5B_PROX_1_ON;

// NETWORK 16
_w5 := RUN_REV_TO_GL5B_BIT AND PROX_1_SEEN_AT_GL5B AND PROX_2_SEEN_AT_GL5B;
RUN_REV_TO_GL5B_BIT R= _w5;
GVL_CONVEYORS.GL2.At_GL5B S= _w5;

// NETWORK 17
_w6 := NOT RUN_REV_TO_GL5B_BIT AND NOT GVL_CONVEYORS.GL2.AT_GL5B_PROX_1_ON AND NOT GVL_CONVEYORS.GL2.AT_GL5B_PROX_2_ON;
PROX_2_SEEN_AT_GL5B R= _w6;
GVL_CONVEYORS.GL2.At_GL5B R= _w6;
PROX_1_SEEN_AT_GL5B R= _w6;

// NETWORK 18: // GL2 IS OCCUPIED AT GL5 POSITION AND DOWNSTREAM PART REQUEST WITH DOOR CLOSED. REQUEST DOOR TO OPEN.
GL1_RD.OPEN_REQUEST := GVL_CONVEYORS.GL1.Ok_To_Run AND GVL_CONVEYORS.ALL_CONVEYORS_IN_CYCLE AND (GVL_CONVEYORS.GL2.AT_GL5B_PROX_1_ON AND GVL_CONVEYORS.GL2.AT_GL5B_PROX_2_ON AND GVL_CONVEYORS.GL2.Occupied AND NOT GVL_CONVEYORS.GL1.Moving AND NOT GVL_CONVEYORS.GL2.Moving AND GL1_RD.DOWN_SWITCH_IS_ON AND (GVL_CONVEYORS.GL6.Calling_For_Part OR GVL_CONVEYORS.GL8.Calling_For_Part OR GVL_CONVEYORS.GL2.Calling_For_Part AND GVL_CONVEYORS.GL2.Moving_to_GL5) OR GL1_RD.OPEN_REQUEST AND NOT GL1_RD.UP_SWITCH_IS_ON);

// NETWORK 19: // SET DOOR STATUS BITS FOR OPEN AND CLOSED
GL1_RD.DOOR_OPEN := GVL_CONVEYORS.GL1.Ok_To_Run AND GVL_CONVEYORS.ALL_CONVEYORS_IN_CYCLE AND GL1_RD.UP_SWITCH_IS_ON;

// NETWORK 20
GL1_RD.DOOR_CLOSED := GVL_CONVEYORS.GL1.Ok_To_Run AND GVL_CONVEYORS.ALL_CONVEYORS_IN_CYCLE AND GL1_RD.DOWN_SWITCH_IS_ON;

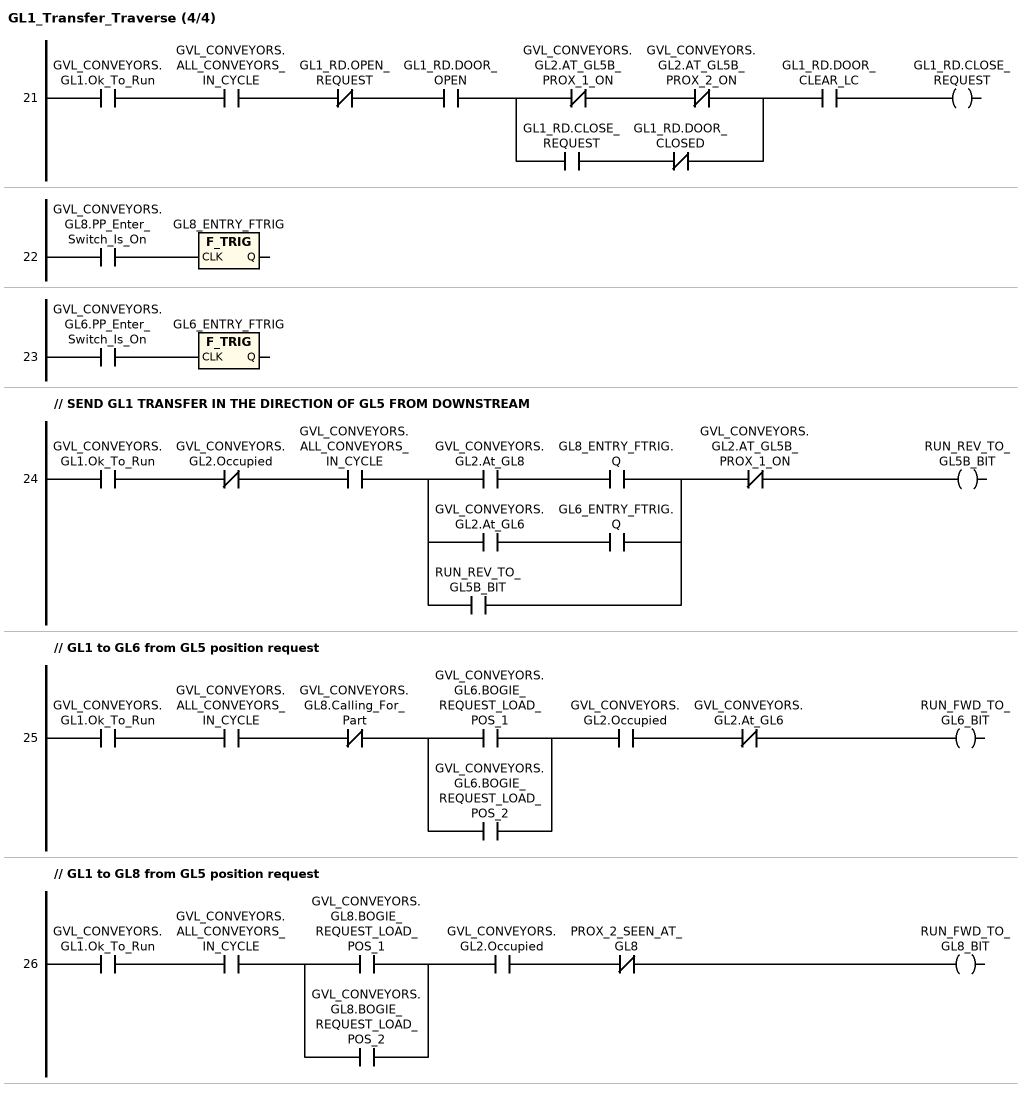
// NETWORK 21
GL1_RD.CLOSE_REQUEST := GVL_CONVEYORS.GL1.Ok_To_Run AND GVL_CONVEYORS.ALL_CONVEYORS_IN_CYCLE AND NOT GL1_RD.OPEN_REQUEST AND GL1_RD.DOOR_OPEN AND (NOT GVL_CONVEYORS.GL2.AT_GL5B_PROX_1_ON AND NOT GVL_CONVEYORS.GL2.AT_GL5B_PROX_2_ON OR GL1_RD.CLOSE_REQUEST AND NOT GL1_RD.DOOR_CLOSED) AND GL1_RD.DOOR_CLEAR_LC;

// NETWORK 22
GL8_ENTRY_FTRIG(CLK := GVL_CONVEYORS.GL8.PP_Enter_Switch_Is_On); // F_TRIG

// NETWORK 23
GL6_ENTRY_FTRIG(CLK := GVL_CONVEYORS.GL6.PP_Enter_Switch_Is_On); // F_TRIG

// NETWORK 24: // SEND GL1 TRANSFER IN THE DIRECTION OF GL5 FROM DOWNSTREAM
RUN_REV_TO_GL5B_BIT := GVL_CONVEYORS.GL1.Ok_To_Run AND NOT GVL_CONVEYORS.GL2.Occupied AND GVL_CONVEYORS.ALL_CONVEYORS_IN_CYCLE AND (GVL_CONVEYORS.GL2.At_GL8 AND GL8_ENTRY_FTRIG.Q OR GVL_CONVEYORS.GL2.At_GL6 AND GL6_ENTRY_FTRIG.Q OR RUN_REV_TO_GL5B_BIT) AND NOT GVL_CONVEYORS.GL2.AT_GL5B_PROX_1_ON;

// NETWORK 25: // GL1 to GL6 from GL5 position request
RUN_FWD_TO_GL6_BIT := GVL_CONVEYORS.GL1.Ok_To_Run AND GVL_CONVEYORS.ALL_CONVEYORS_IN_CYCLE AND NOT GVL_CONVEYORS.GL8.Calling_For_Part AND (GVL_CONVEYORS.GL6.BOGIE_REQUEST_LOAD_POS_1 OR GVL_CONVEYORS.GL6.BOGIE_REQUEST_LOAD_POS_2) AND GVL_CONVEYORS.GL2.Occupied AND NOT GVL_CONVEYORS.GL2.At_GL6;

// NETWORK 26: // GL1 to GL8 from GL5 position request
RUN_FWD_TO_GL8_BIT := GVL_CONVEYORS.GL1.Ok_To_Run AND GVL_CONVEYORS.ALL_CONVEYORS_IN_CYCLE AND (GVL_CONVEYORS.GL8.BOGIE_REQUEST_LOAD_POS_1 OR GVL_CONVEYORS.GL8.BOGIE_REQUEST_LOAD_POS_2) AND GVL_CONVEYORS.GL2.Occupied AND NOT PROX_2_SEEN_AT_GL8;

END_PROGRAM

// ---- Machine System/PRGs/Conveyors/GL10_Transfer_Traverse.TcPOU
PROGRAM GL10_Transfer_Traverse
VAR
	GL10: sTransfer;
	GL11: sTransfer;
	GL12: sTransfer;
	GL3: sConveyor;
	GL7: sConveyor;
	GL9: sConveyor;
	GL10_RD: SRoll_Door;
	GL12_RD: SRoll_Door;
	RUN_FWD_TO_GL3_BIT : BOOL; // GL11 OCCUPIED, GL3 REQUESTING PART, RUN TO GL3 POSITION
	RUN_REV_TO_GL7_BIT : BOOL; // GL11 EMPTY, GL7 REQUESTING PICK UP, RUN TO GL7 POSITION
	RUN_REV_TO_GL9_BIT : BOOL; // GL11 EMPTY, GL9 REQUESTING PICK UP, RUN TO GL9 POSITION
	RUN_REV_TO_GL12_BIT : BOOL; // GL11 EMPTY, GL11 RUN TO GL12 POSITION
END_VAR
VAR // added by the converter: edge detectors and wires of the graphical bodies
    _w1 : BOOL;
END_VAR

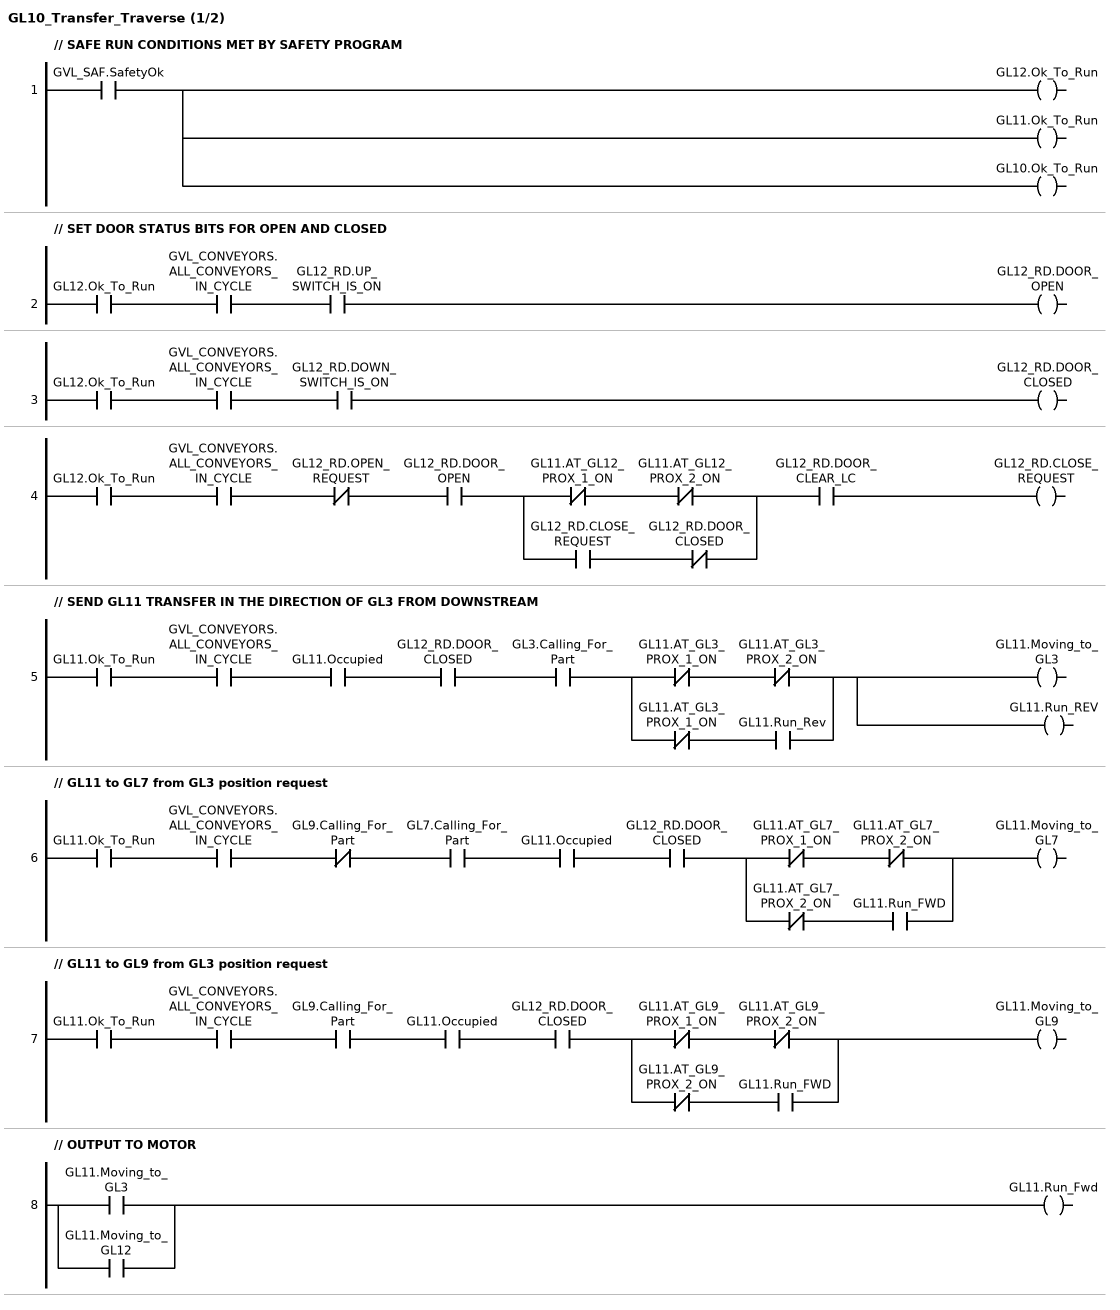
// NETWORK 1: // SAFE RUN CONDITIONS MET BY SAFETY PROGRAM
GL12.Ok_To_Run := GVL_SAF.SafetyOk;
GL11.Ok_To_Run := GVL_SAF.SafetyOk;
GL10.Ok_To_Run := GVL_SAF.SafetyOk;

// NETWORK 2: // SET DOOR STATUS BITS FOR OPEN AND CLOSED
GL12_RD.DOOR_OPEN := GL12.Ok_To_Run AND GVL_CONVEYORS.ALL_CONVEYORS_IN_CYCLE AND GL12_RD.UP_SWITCH_IS_ON;

// NETWORK 3
GL12_RD.DOOR_CLOSED := GL12.Ok_To_Run AND GVL_CONVEYORS.ALL_CONVEYORS_IN_CYCLE AND GL12_RD.DOWN_SWITCH_IS_ON;

// NETWORK 4
GL12_RD.CLOSE_REQUEST := GL12.Ok_To_Run AND GVL_CONVEYORS.ALL_CONVEYORS_IN_CYCLE AND NOT GL12_RD.OPEN_REQUEST AND GL12_RD.DOOR_OPEN AND (NOT GL11.AT_GL12_PROX_1_ON AND NOT GL11.AT_GL12_PROX_2_ON OR GL12_RD.CLOSE_REQUEST AND NOT GL12_RD.DOOR_CLOSED) AND GL12_RD.DOOR_CLEAR_LC;

// NETWORK 5: // SEND GL11 TRANSFER IN THE DIRECTION OF GL3 FROM DOWNSTREAM
_w1 := GL11.Ok_To_Run AND GVL_CONVEYORS.ALL_CONVEYORS_IN_CYCLE AND GL11.Occupied AND GL12_RD.DOOR_CLOSED AND GL3.Calling_For_Part AND (NOT GL11.AT_GL3_PROX_1_ON AND NOT GL11.AT_GL3_PROX_2_ON OR NOT GL11.AT_GL3_PROX_1_ON AND GL11.Run_Rev);
GL11.Moving_to_GL3 := _w1;
GL11.Run_REV := _w1;

// NETWORK 6: // GL11 to GL7 from GL3 position request
GL11.Moving_to_GL7 := GL11.Ok_To_Run AND GVL_CONVEYORS.ALL_CONVEYORS_IN_CYCLE AND NOT GL9.Calling_For_Part AND GL7.Calling_For_Part AND GL11.Occupied AND GL12_RD.DOOR_CLOSED AND (NOT GL11.AT_GL7_PROX_1_ON AND NOT GL11.AT_GL7_PROX_2_ON OR NOT GL11.AT_GL7_PROX_2_ON AND GL11.Run_FWD);

// NETWORK 7: // GL11 to GL9 from GL3 position request
GL11.Moving_to_GL9 := GL11.Ok_To_Run AND GVL_CONVEYORS.ALL_CONVEYORS_IN_CYCLE AND GL9.Calling_For_Part AND GL11.Occupied AND GL12_RD.DOOR_CLOSED AND (NOT GL11.AT_GL9_PROX_1_ON AND NOT GL11.AT_GL9_PROX_2_ON OR NOT GL11.AT_GL9_PROX_2_ON AND GL11.Run_FWD);

// NETWORK 8: // OUTPUT TO MOTOR
GL11.Run_Fwd := GL11.Moving_to_GL3 OR GL11.Moving_to_GL12;

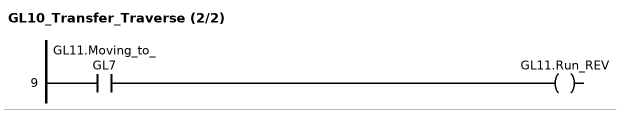
// NETWORK 9
GL11.Run_REV := GL11.Moving_to_GL7;

END_PROGRAM

// ---- Machine System/PRGs/Conveyors/GL11_Transfer.TcPOU
PROGRAM GL11_Transfer
VAR
	GL11: sTransfer;
	GL3: sConveyor;
	GL7: sConveyor;
	GL9: sConveyor;
	GL12: sConveyor;
	GL1_RD: SRoll_Door;
	GL11_PASSSED_ROLL_DOOR : BOOL;
	RUN_FWD_TO_GL3_BIT : BOOL; // GL11 OCCUPIED, GL3 REQUESTING PART, RUN TO GL3 POSITION
	RUN_REV_TO_GL11_BIT : BOOL; //GL11 EMPTY, GL7 OR GL8 REQUESTING PICK UP
	CASE_STOP_UP_REQUEST : BOOL;
END_VAR

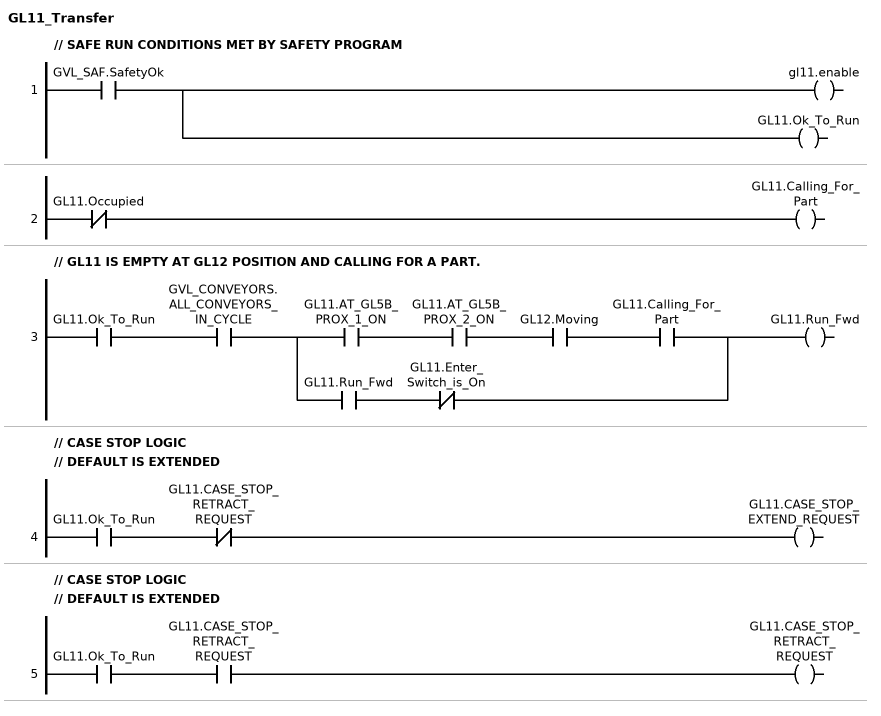
// NETWORK 1: // SAFE RUN CONDITIONS MET BY SAFETY PROGRAM
gl11.enable := GVL_SAF.SafetyOk;
GL11.Ok_To_Run := GVL_SAF.SafetyOk;

// NETWORK 2
GL11.Calling_For_Part := NOT GL11.Occupied;

// NETWORK 3: // GL11 IS EMPTY AT GL12 POSITION AND CALLING FOR A PART.
GL11.Run_Fwd := GL11.Ok_To_Run AND GVL_CONVEYORS.ALL_CONVEYORS_IN_CYCLE AND (GL11.AT_GL5B_PROX_1_ON AND GL11.AT_GL5B_PROX_2_ON AND GL12.Moving AND GL11.Calling_For_Part OR GL11.Run_Fwd AND NOT GL11.Enter_Switch_is_On);

// NETWORK 4: // CASE STOP LOGIC // DEFAULT IS EXTENDED
GL11.CASE_STOP_EXTEND_REQUEST := GL11.Ok_To_Run AND NOT GL11.CASE_STOP_RETRACT_REQUEST;

// NETWORK 5: // CASE STOP LOGIC // DEFAULT IS EXTENDED
GL11.CASE_STOP_RETRACT_REQUEST := GL11.Ok_To_Run AND GL11.CASE_STOP_RETRACT_REQUEST;

END_PROGRAM

// ---- Machine System/PRGs/Conveyors/GL2_Transfer.TcPOU
PROGRAM GL2_Transfer
VAR
	
	
	GL1_RD: SRoll_Door;
	GL2_PASSSED_ROLL_DOOR : BOOL;
	RUN_FWD_TO_GL6_BIT : BOOL; // GL2 OCCUPIED, GL6 REQUESTING PART, RUN TO GL6 POSITION
	RUN_FWD_TO_GL8_BIT : BOOL; // GL2 OCCUPIED, GL8 REQUESTING PART, RUN TO GL8 POSITION
	RUN_REV_TO_GL5_BIT : BOOL; //GL2 EMPTY, GL2 REQUESTING PART, RUN TO GL5 POSITION
	TOF_occupied_delay_off: tof;
	TOF_occupied_delay_of_elapsed: TIME;
	
END_VAR
VAR // added by the converter: edge detectors and wires of the graphical bodies
    _w1 : BOOL;
END_VAR

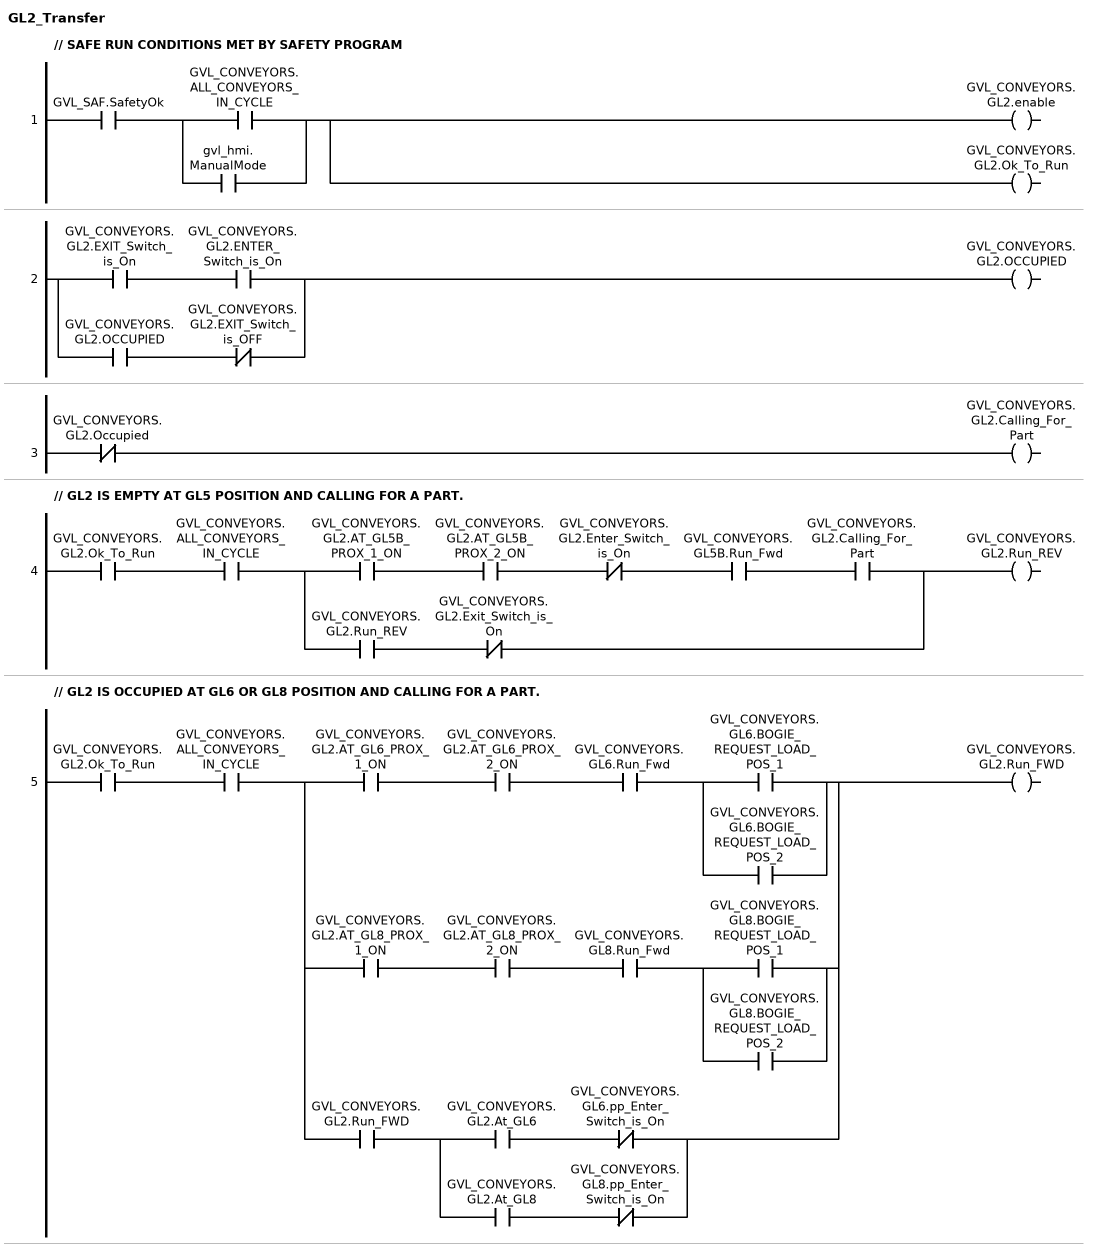
// NETWORK 1: // SAFE RUN CONDITIONS MET BY SAFETY PROGRAM
_w1 := GVL_SAF.SafetyOk AND (GVL_CONVEYORS.ALL_CONVEYORS_IN_CYCLE OR gvl_hmi.ManualMode);
GVL_CONVEYORS.GL2.enable := _w1;
GVL_CONVEYORS.GL2.Ok_To_Run := _w1;

// NETWORK 2
GVL_CONVEYORS.GL2.OCCUPIED := GVL_CONVEYORS.GL2.EXIT_Switch_is_On AND GVL_CONVEYORS.GL2.ENTER_Switch_is_On OR GVL_CONVEYORS.GL2.OCCUPIED AND NOT GVL_CONVEYORS.GL2.EXIT_Switch_is_OFF;

// NETWORK 3
GVL_CONVEYORS.GL2.Calling_For_Part := NOT GVL_CONVEYORS.GL2.Occupied;

// NETWORK 4: // GL2 IS EMPTY AT GL5 POSITION AND CALLING FOR A PART.
GVL_CONVEYORS.GL2.Run_REV := GVL_CONVEYORS.GL2.Ok_To_Run AND GVL_CONVEYORS.ALL_CONVEYORS_IN_CYCLE AND (GVL_CONVEYORS.GL2.AT_GL5B_PROX_1_ON AND GVL_CONVEYORS.GL2.AT_GL5B_PROX_2_ON AND NOT GVL_CONVEYORS.GL2.Enter_Switch_is_On AND GVL_CONVEYORS.GL5B.Run_Fwd AND GVL_CONVEYORS.GL2.Calling_For_Part OR GVL_CONVEYORS.GL2.Run_REV AND NOT GVL_CONVEYORS.GL2.Exit_Switch_is_On);

// NETWORK 5: // GL2 IS OCCUPIED AT GL6 OR GL8 POSITION AND CALLING FOR A PART.
GVL_CONVEYORS.GL2.Run_FWD := GVL_CONVEYORS.GL2.Ok_To_Run AND GVL_CONVEYORS.ALL_CONVEYORS_IN_CYCLE AND (GVL_CONVEYORS.GL2.AT_GL6_PROX_1_ON AND GVL_CONVEYORS.GL2.AT_GL6_PROX_2_ON AND GVL_CONVEYORS.GL6.Run_Fwd AND (GVL_CONVEYORS.GL6.BOGIE_REQUEST_LOAD_POS_1 OR GVL_CONVEYORS.GL6.BOGIE_REQUEST_LOAD_POS_2) OR GVL_CONVEYORS.GL2.AT_GL8_PROX_1_ON AND GVL_CONVEYORS.GL2.AT_GL8_PROX_2_ON AND GVL_CONVEYORS.GL8.Run_Fwd AND (GVL_CONVEYORS.GL8.BOGIE_REQUEST_LOAD_POS_1 OR GVL_CONVEYORS.GL8.BOGIE_REQUEST_LOAD_POS_2) OR GVL_CONVEYORS.GL2.Run_FWD AND (GVL_CONVEYORS.GL2.At_GL6 AND NOT GVL_CONVEYORS.GL6.pp_Enter_Switch_is_On OR GVL_CONVEYORS.GL2.At_GL8 AND NOT GVL_CONVEYORS.GL8.pp_Enter_Switch_is_On));

END_PROGRAM

// ---- Machine System/PRGs/Conveyors/GL3_Accumulation.TcPOU
PROGRAM GL3_Accumulation
VAR
	
	RUN_FWD_TO_GL4_BIT : BOOL; // GL4 EMPTY SO SEND PART FROM GL3 TO GL4
	RUN_FWD_TO_EXIT_BIT : BOOL; // RUN GL3 FWD TO EXIT SENSOR
	GL4_ENTRY_FTRIG:  F_TRIG;
	
END_VAR
VAR // added by the converter: edge detectors and wires of the graphical bodies
    _w1 : BOOL;
END_VAR

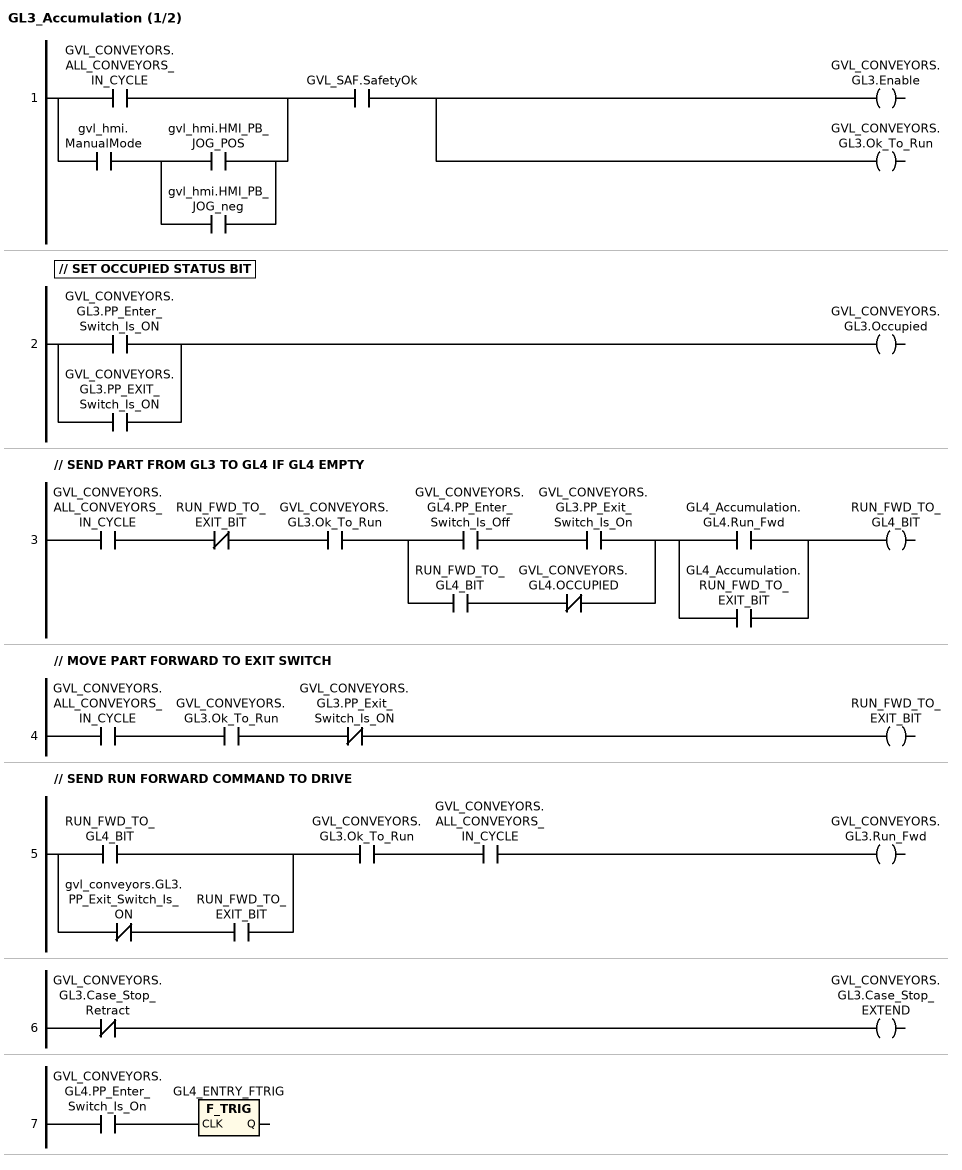
// NETWORK 1
_w1 := (GVL_CONVEYORS.ALL_CONVEYORS_IN_CYCLE OR gvl_hmi.ManualMode AND (gvl_hmi.HMI_PB_JOG_POS OR gvl_hmi.HMI_PB_JOG_neg)) AND GVL_SAF.SafetyOk;
GVL_CONVEYORS.GL3.Enable := _w1;
GVL_CONVEYORS.GL3.Ok_To_Run := _w1;

// NETWORK 2
// label: // SET OCCUPIED STATUS BIT
GVL_CONVEYORS.GL3.Occupied := GVL_CONVEYORS.GL3.PP_Enter_Switch_Is_ON OR GVL_CONVEYORS.GL3.PP_EXIT_Switch_Is_ON;

// NETWORK 3: // SEND PART FROM GL3 TO GL4 IF GL4 EMPTY
RUN_FWD_TO_GL4_BIT := GVL_CONVEYORS.ALL_CONVEYORS_IN_CYCLE AND NOT RUN_FWD_TO_EXIT_BIT AND GVL_CONVEYORS.GL3.Ok_To_Run AND (GVL_CONVEYORS.GL4.PP_Enter_Switch_Is_Off AND GVL_CONVEYORS.GL3.PP_Exit_Switch_Is_On OR RUN_FWD_TO_GL4_BIT AND NOT GVL_CONVEYORS.GL4.OCCUPIED) AND (GL4_Accumulation.GL4.Run_Fwd OR GL4_Accumulation.RUN_FWD_TO_EXIT_BIT);

// NETWORK 4: // MOVE PART FORWARD TO EXIT SWITCH
RUN_FWD_TO_EXIT_BIT := GVL_CONVEYORS.ALL_CONVEYORS_IN_CYCLE AND GVL_CONVEYORS.GL3.Ok_To_Run AND NOT GVL_CONVEYORS.GL3.PP_Exit_Switch_Is_ON;

// NETWORK 5: // SEND RUN FORWARD COMMAND TO DRIVE
GVL_CONVEYORS.GL3.Run_Fwd := (RUN_FWD_TO_GL4_BIT OR NOT gvl_conveyors.GL3.PP_Exit_Switch_Is_ON AND RUN_FWD_TO_EXIT_BIT) AND GVL_CONVEYORS.GL3.Ok_To_Run AND GVL_CONVEYORS.ALL_CONVEYORS_IN_CYCLE;

// NETWORK 6
GVL_CONVEYORS.GL3.Case_Stop_EXTEND := NOT GVL_CONVEYORS.GL3.Case_Stop_Retract;

// NETWORK 7
GL4_ENTRY_FTRIG(CLK := GVL_CONVEYORS.GL4.PP_Enter_Switch_Is_On); // F_TRIG

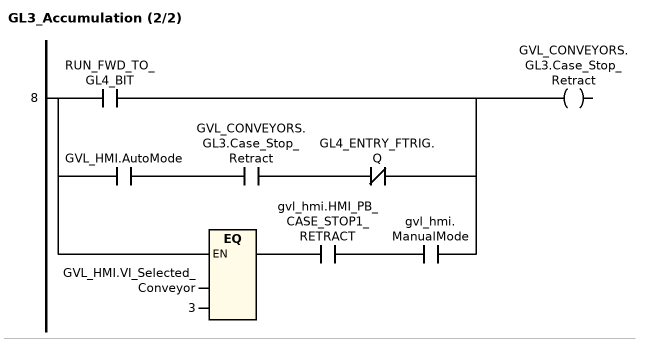
// NETWORK 8
GVL_CONVEYORS.GL3.Case_Stop_Retract := RUN_FWD_TO_GL4_BIT OR GVL_HMI.AutoMode AND GVL_CONVEYORS.GL3.Case_Stop_Retract AND NOT GL4_ENTRY_FTRIG.Q OR GVL_HMI.VI_Selected_Conveyor = 3 AND gvl_hmi.HMI_PB_CASE_STOP1_RETRACT AND gvl_hmi.ManualMode;

END_PROGRAM

// ---- Machine System/PRGs/Conveyors/GL4_Accumulation.TcPOU
PROGRAM GL4_Accumulation
VAR
	GL4: sConveyor;
	GL5: sConveyor;
	RUN_FWD_TO_GL5A_BIT : BOOL; // GL5 EMPTY SO SEND PART FROM GL4 TO GL5
	RUN_FWD_TO_EXIT_BIT : BOOL; // RUN GL4 FWD TO EXIT SENSOR
	GL5A_ENTRY_FTRIG:  F_TRIG;
	
	TEST: BOOL;
END_VAR
VAR // added by the converter: edge detectors and wires of the graphical bodies
    _w1 : BOOL;
END_VAR

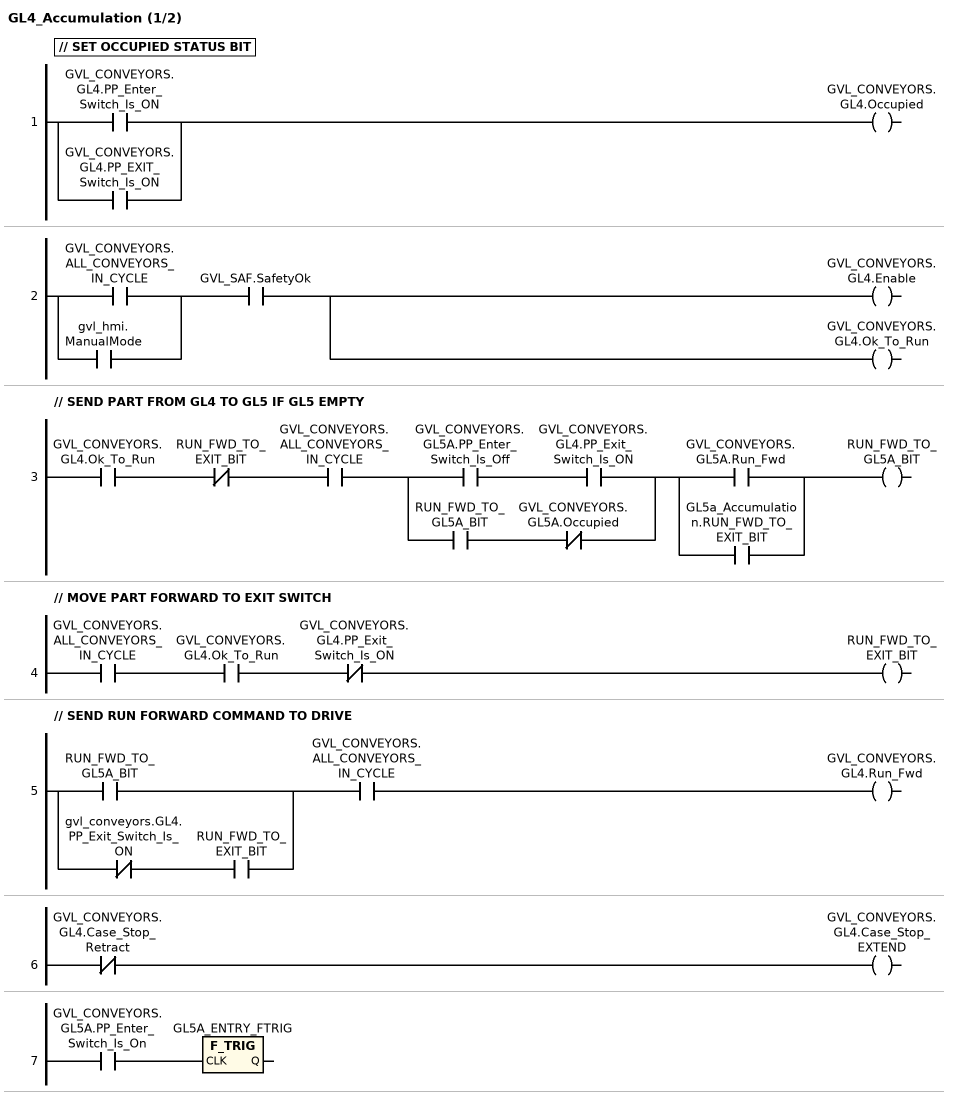
// NETWORK 1
// label: // SET OCCUPIED STATUS BIT
GVL_CONVEYORS.GL4.Occupied := GVL_CONVEYORS.GL4.PP_Enter_Switch_Is_ON OR GVL_CONVEYORS.GL4.PP_EXIT_Switch_Is_ON;

// NETWORK 2
_w1 := (GVL_CONVEYORS.ALL_CONVEYORS_IN_CYCLE OR gvl_hmi.ManualMode) AND GVL_SAF.SafetyOk;
GVL_CONVEYORS.GL4.Enable := _w1;
GVL_CONVEYORS.GL4.Ok_To_Run := _w1;

// NETWORK 3: // SEND PART FROM GL4 TO GL5 IF GL5 EMPTY
RUN_FWD_TO_GL5A_BIT := GVL_CONVEYORS.GL4.Ok_To_Run AND NOT RUN_FWD_TO_EXIT_BIT AND GVL_CONVEYORS.ALL_CONVEYORS_IN_CYCLE AND (GVL_CONVEYORS.GL5A.PP_Enter_Switch_Is_Off AND GVL_CONVEYORS.GL4.PP_Exit_Switch_Is_ON OR RUN_FWD_TO_GL5A_BIT AND NOT GVL_CONVEYORS.GL5A.Occupied) AND (GVL_CONVEYORS.GL5A.Run_Fwd OR GL5a_Accumulation.RUN_FWD_TO_EXIT_BIT);

// NETWORK 4: // MOVE PART FORWARD TO EXIT SWITCH
RUN_FWD_TO_EXIT_BIT := GVL_CONVEYORS.ALL_CONVEYORS_IN_CYCLE AND GVL_CONVEYORS.GL4.Ok_To_Run AND NOT GVL_CONVEYORS.GL4.PP_Exit_Switch_Is_ON;

// NETWORK 5: // SEND RUN FORWARD COMMAND TO DRIVE
GVL_CONVEYORS.GL4.Run_Fwd := (RUN_FWD_TO_GL5A_BIT OR NOT gvl_conveyors.GL4.PP_Exit_Switch_Is_ON AND RUN_FWD_TO_EXIT_BIT) AND GVL_CONVEYORS.ALL_CONVEYORS_IN_CYCLE;

// NETWORK 6
GVL_CONVEYORS.GL4.Case_Stop_EXTEND := NOT GVL_CONVEYORS.GL4.Case_Stop_Retract;

// NETWORK 7
GL5A_ENTRY_FTRIG(CLK := GVL_CONVEYORS.GL5A.PP_Enter_Switch_Is_On); // F_TRIG

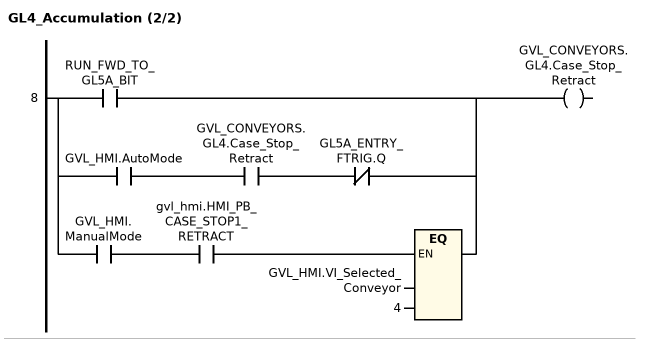
// NETWORK 8
GVL_CONVEYORS.GL4.Case_Stop_Retract := RUN_FWD_TO_GL5A_BIT OR GVL_HMI.AutoMode AND GVL_CONVEYORS.GL4.Case_Stop_Retract AND NOT GL5A_ENTRY_FTRIG.Q OR GVL_HMI.ManualMode AND gvl_hmi.HMI_PB_CASE_STOP1_RETRACT AND GVL_HMI.VI_Selected_Conveyor = 4;

END_PROGRAM

// ---- Machine System/PRGs/Conveyors/GL5A_Accumulation.TcPOU
PROGRAM GL5A_Accumulation
VAR
	
	RUN_FWD_TO_GL5B_BIT : BOOL; // GL2 EMPTY SO SEND PART FROM GL5 TO GL2
	RUN_FWD_TO_EXIT_BIT : BOOL; // RUN GL5 FWD TO EXIT SENSOR
	
	GL5B_ENTRY_FTRIG:  F_TRIG;
END_VAR
VAR // added by the converter: edge detectors and wires of the graphical bodies
    _w1 : BOOL;
END_VAR

